	{attribute 'TcIecLibraryType'}
	{attribute 'external_name' := 'F_VN_RegionOrientationExp_GUID_B2683D61_49B5_467D_FA98_13B80F80665C'}
	(* Calculate the orientation of a region based on a binary image that contains a non zero value for every pixel in that region. (expert function) *)
	FUNCTION F_VN_RegionOrientationExp : HRESULT
	VAR_INPUT
		ipSrcImage	:	ITcVnImage;	(* Source image (1 channel, binary) *)
	END_VAR
	VAR_IN_OUT
		stOrientation	:	TcVnRotatedRectangle;	(* Resulting rotated rectangle, containig center of mass, lenghts of axes, and rotation angle of the region in clockwise direction. *)
	END_VAR
	VAR_INPUT
		eMethod	:	ETcVnOrientationMethod;	(* Method for calculating the orientation. *)
		hrPrev	:	HRESULT;	(* HRESULT indicating the result of previous operations (If SUCCEEDED(hrPrev) equals false, no operation is executed.) *)
	END_VAR

END_FUNCTION

// Functions/Measurement/F_VN_AdjustSearchWindowOrientationToLinearEdge

	{attribute 'TcIecLibraryType'}
	{attribute 'external_name' := 'F_VN_AdjustSearchWindowOrientationToLinearEdge_GUID_4BF80E17_9DF4_4449_FA19_D076489CDE34'}
	(* Adjust the search window to be orthogonal to a linear edge. Might be helpful before calling edge localization and distance measurement functions that rely on the search window. *)
	FUNCTION F_VN_AdjustSearchWindowOrientationToLinearEdge : HRESULT
	VAR_INPUT
		ipSrcImage	:	ITcVnImage;	(* Source image *)
	END_VAR
	VAR_IN_OUT
		aStartPoint	:	TcVnPoint2_REAL;	(* Position from which to start the search process (in the direction of aEndPoint), which is not changed *)
		aEndPoint	:	TcVnPoint2_REAL;	(* Position where the search process ends, which is adjusted by this function *)
	END_VAR
	VAR_INPUT
		eEdgeDirection	:	ETcVnEdgeDirection;	(* Specification of the edge direction to search for *)
		fMinStrength	:	REAL;	(* Specification of the minimum strength (intensity difference) of the edge to search for *)
		nMaxThickness	:	UDINT;	(* Specification of the maximum thickness of the edge to search for, which means fMinStrength must be reached within nMaxThickness pixels *)
		nSearchLines	:	UDINT;	(* Width of the search window, i.e. the number of search lines (3, 5, 7, ...), centered around the line specified by aStartPoint and aEndPoint *)
		hrPrev	:	HRESULT;	(* HRESULT indicating the result of previous operations (If SUCCEEDED(hrPrev) equals false, no operation is executed.) *)
	END_VAR

END_FUNCTION

// Functions/Measurement/F_VN_ClosestPointsBF

	{attribute 'TcIecLibraryType'}
	{attribute 'external_name' := 'F_VN_ClosestPointsBF_GUID_F8745723_FA66_485A_C6BC_8B3A81941337'}
	(* Find the closest distance between two 2d point sets of the same type, using a brute force approach. *)
	FUNCTION F_VN_ClosestPointsBF : HRESULT
	VAR_INPUT
		ipPointSet1	:	ITcVnContainer;	(* Container with 1st set of 2d points *)
		ipPointSet2	:	ITcVnContainer;	(* Container with 2nd set of 2d points *)
	END_VAR
	VAR_IN_OUT
		fMinDist	:	LREAL;	(* Returns the minimum distance between 2 points of the different point sets *)
		aPoint1	:	TcVnPoint2_LREAL;	(* Returns the point out of ipPointSet1, for which fMinDist is achieved *)
		aPoint2	:	TcVnPoint2_LREAL;	(* Returns the point out of ipPointSet2, for which fMinDist is achieved *)
	END_VAR
	VAR_INPUT
		hrPrev	:	HRESULT;	(* HRESULT indicating the result of previous operations (If SUCCEEDED(hrPrev) equals false, no operation is executed.) *)
	END_VAR

END_FUNCTION

// Functions/Measurement/F_VN_LocateCircularArc

	{attribute 'TcIecLibraryType'}
	{attribute 'external_name' := 'F_VN_LocateCircularArc_GUID_5C99AC69_8B36_49C3_F767_A0447ABA5FEC'}
	(* Locate a circular arc, using an interpolation method. *)
	FUNCTION F_VN_LocateCircularArc : HRESULT
	VAR_INPUT
		ipSrcImage	:	ITcVnImage;	(* Source image (1 channel) *)
	END_VAR
	VAR_IN_OUT
		stCircularArc	:	TcVnCircularArc;	(* Returns the circular arc parameters *)
		aCenter	:	TcVnPoint2_REAL;	(* Input estimated circle center (only used as a starting point to search for the circle contour, not used for the circle center estimation) *)
	END_VAR
	VAR_INPUT
		fSearchRadius	:	REAL;	(* Input search radius (starting from aCenter, should be greater than the actual circle radius but aCenter + fSearchRadius should be within the image borders) *)
		fArcDirectionRad	:	LREAL;	(* Input search starting direction in radian. Valid range is [-pi, +pi], where right is 0 rad, top is -pi/2 rad and bottom +pi/2 rad. The circular arc should at least be valid in range fArcDirectionRad +- 0.4 rad. *)
		eEdgeDirection	:	ETcVnEdgeDirection;	(* Specification of the edge direction to search for *)
		fMinStrength	:	REAL;	(* Specification of the minimum strength (intensity difference) of the edge to search for *)
		hrPrev	:	HRESULT;	(* HRESULT indicating the result of previous operations (If SUCCEEDED(hrPrev) equals false, no operation is executed.) *)
	END_VAR

END_FUNCTION

// Functions/Measurement/F_VN_LocateCircularArcExp

	{attribute 'TcIecLibraryType'}
	{attribute 'external_name' := 'F_VN_LocateCircularArcExp_GUID_D2973620_C78E_45B3_C257_FC79FEFA4F95'}
	(* Locate a circular arc. (expert function) *)
	FUNCTION F_VN_LocateCircularArcExp : HRESULT
	VAR_INPUT
		ipSrcImage	:	ITcVnImage;	(* Source image (1 channel) *)
	END_VAR
	VAR_IN_OUT
		stCircularArc	:	TcVnCircularArc;	(* Returns the circular arc parameters *)
		aCenter	:	TcVnPoint2_REAL;	(* Input estimated circle center (only used as a starting point to search for the circle contour, not used for the circle center estimation) *)
	END_VAR
	VAR_INPUT
		fSearchRadius	:	REAL;	(* Input search radius (starting from aCenter, should be greater than the actual circle radius but aCenter + fSearchRadius should be within the image borders) *)
		fArcDirectionRad	:	LREAL;	(* Input search starting direction in radian. Valid range is [-pi, +pi], where right is 0 rad, top is -pi/2 rad and bottom +pi/2 rad. The circular arc should at least be valid in range fArcDirectionRad +- 4 * fAngleStepRad) *)
		eEdgeDirection	:	ETcVnEdgeDirection;	(* Specification of the edge direction to search for *)
		fMinStrength	:	REAL;	(* Specification of the minimum strength (intensity difference) of the edge to search for *)
		fAngleStepRad	:	LREAL;	(* Search step in rad (should be chosen so that about 20 - 60 steps are available for the whole arc. In most cases 0.1 rad (5.7 deg) is a good value) *)
		nMaxThickness	:	UDINT;	(* Specification of the maximum thickness of the edge to search for, which means fMinStrength must be reached within nMaxThickness pixels *)
		bInvertSearchDirection	:	BOOL;	(* If true, the search starts from outside the circular arc in direction of the center *)
		nSubpixelsIterations	:	UDINT;	(* Specifies the number of subpixels (for INTERPOLATION, 10 - 20 usually is sufficient) or maximum number of iterations for optimizing the parameters (for APPROX_ERF and APPROX_GAUSSIAN, 50 - 100 usually is sufficient) *)
		fApproxPrecision	:	REAL;	(* Specifies the approximation precision for APPROX_ERF and APPROX_GAUSSIAN (0.001 usually is sufficient, unused for INTERPOLATION) *)
		eAlgorithm	:	ETcVnEdgeDetectionAlgorithm;	(* Selection of the edge detection algorithm *)
		ipContourPoints	:	REFERENCE TO ITcVnContainer;	(* Returns the subpixel accurate contour (optional, set to 0 if not required; ContainerType_Vector_TcVnPoint2_REAL; Non-zero interface pointers are reused.) *)
		hrPrev	:	HRESULT;	(* HRESULT indicating the result of previous operations (If SUCCEEDED(hrPrev) equals false, no operation is executed.) *)
	END_VAR

END_FUNCTION

// Functions/Measurement/F_VN_LocateEdge

	{attribute 'TcIecLibraryType'}
	{attribute 'external_name' := 'F_VN_LocateEdge_GUID_6D658DBC_9003_460D_D8DC_4EA5DD496210'}
	(* Locate the points of the first occuring edge inside a specified search window, using an interpolation method. *)
	FUNCTION F_VN_LocateEdge : HRESULT
	VAR_INPUT
		ipSrcImage	:	ITcVnImage;	(* Source image (1 channel) *)
		ipEdgePoints	:	REFERENCE TO ITcVnContainer;	(* Returns the detected edge points (ContainerType_Vector_TcVnPoint2_REAL) *)
	END_VAR
	VAR_IN_OUT
		aStartPoint	:	TcVnPoint2_REAL;	(* Position from which to start the search process (in the direction of aEndPoint) *)
		aEndPoint	:	TcVnPoint2_REAL;	(* Position where the search process ends *)
	END_VAR
	VAR_INPUT
		eEdgeDirection	:	ETcVnEdgeDirection;	(* Specification of the edge direction to search for *)
		fMinStrength	:	REAL;	(* Specification of the minimum strength (intensity difference) of the edge to search for *)
		nSearchLines	:	UDINT;	(* Width of the search window, i.e. the number of search lines (1, 3, 5, 7, ...), centered around the line specified by aStartPoint and aEndPoint *)
		hrPrev	:	HRESULT;	(* HRESULT indicating the result of previous operations (If SUCCEEDED(hrPrev) equals false, no operation is executed.) *)
	END_VAR
	VAR_OUTPUT
		fAvgStrength	:	REAL;	(* Returns the average strength of the detected edge *)
	END_VAR

END_FUNCTION

// Functions/Measurement/F_VN_LocateEdgeExp

	{attribute 'TcIecLibraryType'}
	{attribute 'external_name' := 'F_VN_LocateEdgeExp_GUID_71867877_E50C_46F9_ECC5_1606F0E48315'}
	(* Locate the points of the first occuring edge inside a specified search window with subpixel accuracy. (expert function) *)
	FUNCTION F_VN_LocateEdgeExp : HRESULT
	VAR_INPUT
		ipSrcImage	:	ITcVnImage;	(* Source image (1 channel) *)
		ipEdgePoints	:	REFERENCE TO ITcVnContainer;	(* Returns the detected edge points (ContainerType_Vector_TcVnPoint2_REAL) *)
	END_VAR
	VAR_IN_OUT
		aStartPoint	:	TcVnPoint2_REAL;	(* Position from which to start the search process (in the direction of aEndPoint) *)
		aEndPoint	:	TcVnPoint2_REAL;	(* Position where the search process ends *)
	END_VAR
	VAR_INPUT
		eEdgeDirection	:	ETcVnEdgeDirection;	(* Specification of the edge direction to search for *)
		fMinStrength	:	REAL;	(* Specification of the minimum strength (intensity difference) of the edge to search for *)
		nSearchLines	:	UDINT;	(* Width of the search window, i.e. the number of search lines (1, 3, 5, 7, ...), centered around the line specified by aStartPoint and aEndPoint *)
		fSearchLineDist	:	REAL;	(* Distance between the search lines in pixels (> 0) *)
		nMaxThickness	:	UDINT;	(* Specification of the maximum thickness of the edge to search for, which means fMinStrength must be reached within nMaxThickness pixels *)
		nSubpixelsIterations	:	UDINT;	(* Specifies the number of subpixels (for INTERPOLATION, 10 - 20 usually is sufficient) or maximum number of iterations for optimizing the parameters (for APPROX_ERF and APPROX_GAUSSIAN, 50 - 100 usually is sufficient) *)
		fApproxPrecision	:	REAL;	(* Specifies the approximation precision for APPROX_ERF and APPROX_GAUSSIAN (0.001 usually is sufficient, unused for INTERPOLATION) *)
		eAlgorithm	:	ETcVnEdgeDetectionAlgorithm;	(* Selection of the edge detection algorithm *)
		hrPrev	:	HRESULT;	(* HRESULT indicating the result of previous operations (If SUCCEEDED(hrPrev) equals false, no operation is executed.) *)
	END_VAR
	VAR_OUTPUT
		fAvgStrength	:	REAL;	(* Returns the average strength of the detected edge *)
	END_VAR

END_FUNCTION

// Functions/Measurement/F_VN_LocateEdges

	{attribute 'TcIecLibraryType'}
	{attribute 'external_name' := 'F_VN_LocateEdges_GUID_16CD5812_FF7D_41F8_D2D0_ABD474139878'}
	(* Locate the points of multiple occuring edges inside a specified search window, using an interpolation method. *)
	FUNCTION F_VN_LocateEdges : HRESULT
	VAR_INPUT
		ipSrcImage	:	ITcVnImage;	(* Source image (1 channel) *)
		ipEdgePoints	:	REFERENCE TO ITcVnContainer;	(* Returns the detected edge points (ContainerType_Vector_Vector_TcVnPoint2_REAL) *)
	END_VAR
	VAR_IN_OUT
		aStartPoint	:	TcVnPoint2_REAL;	(* Position from which to start the search process (in the direction of aEndPoint) *)
		aEndPoint	:	TcVnPoint2_REAL;	(* Position where the search process ends *)
	END_VAR
	VAR_INPUT
		nNumEdges	:	UDINT;	(* The (maximum) number of edges to search for *)
		eEdgeDirection	:	ETcVnEdgeDirection;	(* Specification of the edge direction to search for *)
		bAlternateDirection	:	BOOL;	(* If true, eEdgeDirection is alternated after each detected edge. Else, only edges with eEdgeDirection are searched for. *)
		fMinStrength	:	REAL;	(* Specification of the minimum strength (intensity difference) of the edge to search for *)
		nSearchLines	:	UDINT;	(* Width of the search window, i.e. the number of search lines (1, 3, 5, 7, ...), centered around the line specified by aStartPoint and aEndPoint *)
		hrPrev	:	HRESULT;	(* HRESULT indicating the result of previous operations (If SUCCEEDED(hrPrev) equals false, no operation is executed.) *)
	END_VAR
	VAR_OUTPUT
		fAvgStrength	:	REAL;	(* Returns the average strength of the detected edges *)
	END_VAR

END_FUNCTION

// Functions/Measurement/F_VN_LocateEdgesExp

	{attribute 'TcIecLibraryType'}
	{attribute 'external_name' := 'F_VN_LocateEdgesExp_GUID_24AB17DE_4502_4635_E826_7D952681F995'}
	(* Locate the points of multiple occuring edges inside a specified search window with subpixel accuracy. (expert function) *)
	FUNCTION F_VN_LocateEdgesExp : HRESULT
	VAR_INPUT
		ipSrcImage	:	ITcVnImage;	(* Source image (1 channel) *)
		ipEdgePoints	:	REFERENCE TO ITcVnContainer;	(* Returns the detected edge points (ContainerType_Vector_Vector_TcVnPoint2_REAL) *)
	END_VAR
	VAR_IN_OUT
		aStartPoint	:	TcVnPoint2_REAL;	(* Position from which to start the search process (in the direction of aEndPoint) *)
		aEndPoint	:	TcVnPoint2_REAL;	(* Position where the search process ends *)
	END_VAR
	VAR_INPUT
		nNumEdges	:	UDINT;	(* The (maximum) number of edges to search for *)
		eEdgeDirection	:	ETcVnEdgeDirection;	(* Specification of the edge direction to search for *)
		bAlternateDirection	:	BOOL;	(* If true, eEdgeDirection is alternated after each detected edge. Else, only edges with eEdgeDirection are searched for. *)
		fMinStrength	:	REAL;	(* Specification of the minimum strength (intensity difference) of the edge to search for *)
		nSearchLines	:	UDINT;	(* Width of the search window, i.e. the number of search lines (1, 3, 5, 7, ...), centered around the line specified by aStartPoint and aEndPoint *)
		fSearchLineDist	:	REAL;	(* Distance between the search lines in pixels (> 0) *)
		nMaxThickness	:	UDINT;	(* Specification of the maximum thickness of the edge to search for, which means fMinStrength must be reached within nMaxThickness pixels *)
		nSubpixelsIterations	:	UDINT;	(* Specifies the number of subpixels (for INTERPOLATION, 10 - 20 usually is sufficient) or maximum number of iterations for optimizing the parameters (for APPROX_ERF and APPROX_GAUSSIAN, 50 - 100 usually is sufficient) *)
		fApproxPrecision	:	REAL;	(* Specifies the approximation precision for APPROX_ERF and APPROX_GAUSSIAN (0.001 usually is sufficient, unused for INTERPOLATION) *)
		eAlgorithm	:	ETcVnEdgeDetectionAlgorithm;	(* Selection of the edge detection algorithm *)
		hrPrev	:	HRESULT;	(* HRESULT indicating the result of previous operations (If SUCCEEDED(hrPrev) equals false, no operation is executed.) *)
	END_VAR
	VAR_OUTPUT
		fAvgStrength	:	REAL;	(* Returns the average strength of the detected edges *)
	END_VAR

END_FUNCTION

// Functions/Measurement/F_VN_LocateEllipse

	{attribute 'TcIecLibraryType'}
	{attribute 'external_name' := 'F_VN_LocateEllipse_GUID_7D53F90F_C5F2_4037_E1F8_744121219137'}
	(* Locate an ellipse, using an interpolation method for locating the edges. *)
	FUNCTION F_VN_LocateEllipse : HRESULT
	VAR_INPUT
		ipSrcImage	:	ITcVnImage;	(* Source image (1 channel) *)
	END_VAR
	VAR_IN_OUT
		stEllipse	:	TcVnRotatedRectangle;	(* Returns the detected ellipse *)
		aCenter	:	TcVnPoint2_REAL;	(* The expected ellipse center *)
	END_VAR
	VAR_INPUT
		fSearchRadius	:	REAL;	(* Radius around aCenter to search for edges (aCenter + fSearchRadius in all directions must be inside image borders!) *)
		eEdgeDirection	:	ETcVnEdgeDirection;	(* Specification of the edge direction to search for (from center to outside ellipse) *)
		fMinStrength	:	REAL;	(* Specification of the minimum strength (intensity difference) of the edge to search for *)
		hrPrev	:	HRESULT;	(* HRESULT indicating the result of previous operations (If SUCCEEDED(hrPrev) equals false, no operation is executed.) *)
	END_VAR

END_FUNCTION

// Functions/Measurement/F_VN_LocateEllipseExp

	{attribute 'TcIecLibraryType'}
	{attribute 'external_name' := 'F_VN_LocateEllipseExp_GUID_0A60BF8D_B9F3_4F5C_FC58_D9258E827D64'}
	(* Locate an ellipse. (expert function) *)
	FUNCTION F_VN_LocateEllipseExp : HRESULT
	VAR_INPUT
		ipSrcImage	:	ITcVnImage;	(* Source image (1 channel) *)
	END_VAR
	VAR_IN_OUT
		stEllipse	:	TcVnRotatedRectangle;	(* Returns the detected ellipse *)
		aCenter	:	TcVnPoint2_REAL;	(* The expected ellipse center *)
	END_VAR
	VAR_INPUT
		fSearchRadius	:	REAL;	(* Radius around aCenter to search for edges *)
		eEdgeDirection	:	ETcVnEdgeDirection;	(* Specification of the edge direction to search for (from center to outside ellipse or other way round, if bInvertSearchDirection is true) *)
		fMinStrength	:	REAL;	(* Specification of the minimum strength (intensity difference) of the edge to search for *)
		nMaxThickness	:	UDINT;	(* Specification of the maximum thickness of the edge to search for, which means fMinStrength must be reached within nMaxThickness pixels *)
		bInvertSearchDirection	:	BOOL;	(* If true, the search starts from outside the ellipse in direction of the center *)
		fMinSearchRadius	:	REAL;	(* Radius around aCenter to skip before starting to search for edges (e.g. to save time or if the center contains edges that should be ignored) *)
		nSubpixelsIterations	:	UDINT;	(* Specifies the number of subpixels (for INTERPOLATION, 10 - 20 usually is sufficient) or maximum number of iterations for optimizing the parameters (for APPROX_ERF and APPROX_GAUSSIAN, 50 - 100 usually is sufficient) *)
		nSearchLines	:	UDINT;	(* Specifies the amount of search lines, which are equally distributed in all directions (must be >= 8 and a multiple of 4) *)
		fApproxPrecision	:	REAL;	(* Specifies the approximation precision for APPROX_ERF and APPROX_GAUSSIAN (0.001 usually is sufficient, unused for INTERPOLATION) *)
		eAlgorithm	:	ETcVnEdgeDetectionAlgorithm;	(* Selection of the edge detection algorithm *)
		ipContourPoints	:	REFERENCE TO ITcVnContainer;	(* Returns the subpixel accurate ellipse contour (optional, set to 0 if not required; ContainerType_Vector_TcVnPoint2_REAL; Non-zero interface pointers are reused.) *)
		hrPrev	:	HRESULT;	(* HRESULT indicating the result of previous operations (If SUCCEEDED(hrPrev) equals false, no operation is executed.) *)
	END_VAR

END_FUNCTION

// Functions/Measurement/F_VN_MeasureAngleBetweenEdges

	{attribute 'TcIecLibraryType'}
	{attribute 'external_name' := 'F_VN_MeasureAngleBetweenEdges_GUID_D045AAF4_339B_4CE5_F178_0EB747DFE41C'}
	(* Measure the angle between 2 edges, using an interpolation method. *)
	FUNCTION F_VN_MeasureAngleBetweenEdges : HRESULT
	VAR_INPUT
		ipSrcImage	:	ITcVnImage;	(* Source image (1 channel) *)
	END_VAR
	VAR_IN_OUT
		fAngle	:	REAL;	(* Returns the angle between the detected edges (radians) *)
		aInnerPoint	:	TcVnPoint2_REAL;	(* Position inside the angle to measure, from which to start the edge search process (in the direction of aOuterPoint1 and aOuterPoint2) *)
		aOuterPoint1	:	TcVnPoint2_REAL;	(* Position where the search process for edge 1 ends *)
		aOuterPoint2	:	TcVnPoint2_REAL;	(* Position where the search process for edge 2 ends *)
	END_VAR
	VAR_INPUT
		eEdgeDirection	:	ETcVnEdgeDirection;	(* Specification of the edge direction from aInnerPoint to aOuterPoint1 and aOuterPoint2 to search for *)
		fMinStrength	:	REAL;	(* Specification of the minimum strength (intensity difference) of the edge to search for *)
		nSearchLines	:	UDINT;	(* Width of the search windows, i.e. the number of search lines (3, 5, 7, ...), centered around the lines specified by aInnerPoint and aOuterPoint1, aOuterPoint2 *)
		hrPrev	:	HRESULT;	(* HRESULT indicating the result of previous operations (If SUCCEEDED(hrPrev) equals false, no operation is executed.) *)
	END_VAR

END_FUNCTION

// Functions/Measurement/F_VN_MeasureAngleBetweenEdgesExp

	{attribute 'TcIecLibraryType'}
	{attribute 'external_name' := 'F_VN_MeasureAngleBetweenEdgesExp_GUID_B9FC8105_DD76_4FBA_C762_CA24E7D135AD'}
	(* Measure the angle between 2 edges. *)
	FUNCTION F_VN_MeasureAngleBetweenEdgesExp : HRESULT
	VAR_INPUT
		ipSrcImage	:	ITcVnImage;	(* Source image (1 channel) *)
	END_VAR
	VAR_IN_OUT
		fAngle	:	REAL;	(* Returns the angle between the detected edges (radians or degrees, depending on bAngleInDegrees) *)
		aInnerPoint	:	TcVnPoint2_REAL;	(* Position inside the angle to measure, from which to start the edge search process (in the direction of aOuterPoint1 and aOuterPoint2) *)
		aOuterPoint1	:	TcVnPoint2_REAL;	(* Position where the search process for edge 1 ends *)
		aOuterPoint2	:	TcVnPoint2_REAL;	(* Position where the search process for edge 2 ends *)
	END_VAR
	VAR_INPUT
		eEdgeDirection	:	ETcVnEdgeDirection;	(* Specification of the edge direction from aInnerPoint to aOuterPoint1 and aOuterPoint2 to search for *)
		fMinStrength	:	REAL;	(* Specification of the minimum strength (intensity difference) of the edge to search for *)
		nSearchLines	:	UDINT;	(* Width of the search window, i.e. the number of search lines (3, 5, 7, ...), centered around the line specified by aInnerPoint and aOuterPoint1, aOuterPoint2 *)
		fSearchLineDist	:	REAL;	(* Distance between the search lines in pixels (> 0) *)
		nMaxThickness	:	UDINT;	(* Specification of the maximum thickness of the edge to search for, which means fMinStrength must be reached within nMaxThickness pixels *)
		bInvertSearchDirection	:	BOOL;	(* If true, the search starts from each aOuterPoint in direction of aInnerPoint *)
		nSubpixelsIterations	:	UDINT;	(* Specifies the number of subpixels (for INTERPOLATION, 10 - 20 usually is sufficient) or maximum number of iterations for optimizing the parameters (for APPROX_ERF and APPROX_GAUSSIAN, 50 - 100 usually is sufficient) *)
		bAngleInDegrees	:	BOOL;	(* fAngle is in degrees, if true *)
		fApproxPrecision	:	REAL;	(* Specifies the approximation precision for APPROX_ERF and APPROX_GAUSSIAN (0.001 usually is sufficient, unused for INTERPOLATION) *)
		eAlgorithm	:	ETcVnEdgeDetectionAlgorithm;	(* Selection of the edge detection algorithm *)
		ipEdgePoints1	:	REFERENCE TO ITcVnContainer;	(* Returns the detected edge points between aInnerPoint and aOuterPoint1 (ContainerType_Vector_TcVnPoint2_REAL) *)
		ipEdgePoints2	:	REFERENCE TO ITcVnContainer;	(* Returns the detected edge points between aInnerPoint and aOuterPoint2 (ContainerType_Vector_TcVnPoint2_REAL) *)
		hrPrev	:	HRESULT;	(* HRESULT indicating the result of previous operations (If SUCCEEDED(hrPrev) equals false, no operation is executed.) *)
	END_VAR

END_FUNCTION

// Functions/Measurement/F_VN_MeasureEdgeDistance

	{attribute 'TcIecLibraryType'}
	{attribute 'external_name' := 'F_VN_MeasureEdgeDistance_GUID_6B314BDA_9727_45F2_FABA_828BF07E8929'}
	(* Measure the distance between 2 parallel edges, using an interpolation method. *)
	FUNCTION F_VN_MeasureEdgeDistance : HRESULT
	VAR_INPUT
		ipSrcImage	:	ITcVnImage;	(* Source image (1 channel) *)
	END_VAR
	VAR_IN_OUT
		fAvgDistance	:	REAL;	(* Returns the average distance between the detected edges *)
		aStartPoint	:	TcVnPoint2_REAL;	(* Position from which to start the search process (in the direction of aEndPoint) *)
		aEndPoint	:	TcVnPoint2_REAL;	(* Position where the search process ends *)
	END_VAR
	VAR_INPUT
		eEdgeDirection	:	ETcVnEdgeDirection;	(* Specification of the edge direction from aStartPoint to aEndPoint to search for *)
		fMinStrength	:	REAL;	(* Specification of the minimum strength (intensity difference) of the edge to search for *)
		nSearchLines	:	UDINT;	(* Width of the search window, i.e. the number of search lines (1, 3, 5, 7, ...), centered around the line specified by aStartPoint and aEndPoint *)
		hrPrev	:	HRESULT;	(* HRESULT indicating the result of previous operations (If SUCCEEDED(hrPrev) equals false, no operation is executed.) *)
	END_VAR

END_FUNCTION

// Functions/Measurement/F_VN_MeasureEdgeDistanceExp

	{attribute 'TcIecLibraryType'}
	{attribute 'external_name' := 'F_VN_MeasureEdgeDistanceExp_GUID_B5A698E0_19B0_4B58_F68B_C2D607FA5C90'}
	(* Measure the distance between 2 parallel edges. (expert function) *)
	FUNCTION F_VN_MeasureEdgeDistanceExp : HRESULT
	VAR_INPUT
		ipSrcImage	:	ITcVnImage;	(* Source image (1 channel) *)
	END_VAR
	VAR_IN_OUT
		fAvgDistance	:	REAL;	(* Returns the average distance between the detected edges *)
		aStartPoint	:	TcVnPoint2_REAL;	(* Position from which to start the search process (in the direction of aEndPoint) *)
		aEndPoint	:	TcVnPoint2_REAL;	(* Position where the search process ends *)
	END_VAR
	VAR_INPUT
		eEdgeDirection	:	ETcVnEdgeDirection;	(* Specification of the edge direction from aStartPoint to aEndPoint to search for *)
		fMinStrength	:	REAL;	(* Specification of the minimum strength (intensity difference) of the edge to search for *)
		nSearchLines	:	UDINT;	(* Width of the search window, i.e. the number of search lines (1, 3, 5, 7, ...), centered around the line specified by aStartPoint and aEndPoint *)
		fSearchLineDist	:	REAL;	(* Distance between the search lines in pixels (> 0) *)
		nMaxThickness	:	UDINT;	(* Specification of the maximum thickness of the edge to search for, which means fMinStrength must be reached within nMaxThickness pixels *)
		bInvertSearchDirection	:	BOOL;	(* If true, the search starts from the center point between aStartPoint and aEndPoint in both directions *)
		fSearchGap	:	REAL;	(* Optional width of a gap (>= 0, centered between aStartPoint and aEndPoint), that is neglected for searching edges (can reduce execution time). The 2 edges to search for must be on different sides of the gap. *)
		nSubpixelsIterations	:	UDINT;	(* Specifies the number of subpixels (for INTERPOLATION, 10 - 20 usually is sufficient) or maximum number of iterations for optimizing the parameters (for APPROX_ERF and APPROX_GAUSSIAN, 50 - 100 usually is sufficient) *)
		fApproxPrecision	:	REAL;	(* Specifies the approximation precision for APPROX_ERF and APPROX_GAUSSIAN (0.001 usually is sufficient, unused for INTERPOLATION) *)
		eAlgorithm	:	ETcVnEdgeDetectionAlgorithm;	(* Selection of the edge detection algorithm *)
		ipEdgePoints1	:	REFERENCE TO ITcVnContainer;	(* Returns the detected edge points of the edge near aStartPoint (optional, set to 0 if not required; ContainerType_Vector_TcVnPoint2_REAL) *)
		ipEdgePoints2	:	REFERENCE TO ITcVnContainer;	(* Returns the detected edge points of the edge near aEndPoint (optional, set to 0 if not required; ContainerType_Vector_TcVnPoint2_REAL) *)
		ipDistances	:	REFERENCE TO ITcVnContainer;	(* Returns the distances between the detected edge points (optional, set to 0 if not required; ContainerType_Vector_REAL) *)
		hrPrev	:	HRESULT;	(* HRESULT indicating the result of previous operations (If SUCCEEDED(hrPrev) equals false, no operation is executed.) *)
	END_VAR

END_FUNCTION

// Functions/Measurement/F_VN_MeasureMinEdgeDistance

	{attribute 'TcIecLibraryType'}
	{attribute 'external_name' := 'F_VN_MeasureMinEdgeDistance_GUID_AD6515FF_4497_4F80_F2EC_1F853CD0ABA8'}
	(* Measure the minimum distance within the specified search window between 2 edges, using an interpolation method. *)
	FUNCTION F_VN_MeasureMinEdgeDistance : HRESULT
	VAR_INPUT
		ipSrcImage	:	ITcVnImage;	(* Source image (1 channel) *)
	END_VAR
	VAR_IN_OUT
		fMinDistance	:	REAL;	(* Returns the minimum distance between the detected edges *)
		aStartPoint	:	TcVnPoint2_REAL;	(* Position from which to start the search process (in the direction of aEndPoint) *)
		aEndPoint	:	TcVnPoint2_REAL;	(* Position where the search process ends *)
	END_VAR
	VAR_INPUT
		eEdgeDirection	:	ETcVnEdgeDirection;	(* Specification of the edge direction from aStartPoint to aEndPoint to search for *)
		fMinStrength	:	REAL;	(* Specification of the minimum strength (intensity difference) of the edge to search for *)
		nSearchLines	:	UDINT;	(* Width of the search window, i.e. the number of search lines (1, 3, 5, 7, ...), centered around the line specified by aStartPoint and aEndPoint *)
		hrPrev	:	HRESULT;	(* HRESULT indicating the result of previous operations (If SUCCEEDED(hrPrev) equals false, no operation is executed.) *)
	END_VAR

END_FUNCTION

// Functions/Measurement/F_VN_MeasureMinEdgeDistanceExp

	{attribute 'TcIecLibraryType'}
	{attribute 'external_name' := 'F_VN_MeasureMinEdgeDistanceExp_GUID_1BC885D6_665A_4846_FCF1_ACE60271C85F'}
	(* Measure the minimum distance within the specified search window between 2 edges. (expert function) *)
	FUNCTION F_VN_MeasureMinEdgeDistanceExp : HRESULT
	VAR_INPUT
		ipSrcImage	:	ITcVnImage;	(* Source image (1 channel) *)
	END_VAR
	VAR_IN_OUT
		fMinDistance	:	REAL;	(* Returns the minimum distance between the detected edges *)
		aStartPoint	:	TcVnPoint2_REAL;	(* Position from which to start the search process (in the direction of aEndPoint) *)
		aEndPoint	:	TcVnPoint2_REAL;	(* Position where the search process ends *)
	END_VAR
	VAR_INPUT
		eEdgeDirection	:	ETcVnEdgeDirection;	(* Specification of the edge direction from aStartPoint to aEndPoint to search for *)
		fMinStrength	:	REAL;	(* Specification of the minimum strength (intensity difference) of the edge to search for *)
		nSearchLines	:	UDINT;	(* Width of the search window, i.e. the number of search lines (1, 3, 5, 7, ...), centered around the line specified by aStartPoint and aEndPoint *)
		fSearchLineDist	:	REAL;	(* Distance between the search lines in pixels (> 0) *)
		nMaxThickness	:	UDINT;	(* Specification of the maximum thickness of the edge to search for, which means fMinStrength must be reached within nMaxThickness pixels *)
		bInvertSearchDirection	:	BOOL;	(* If true, the search starts from the center point between aStartPoint and aEndPoint in both directions *)
		fSearchGap	:	REAL;	(* Optional width of a gap (>= 0, centered between aStartPoint and aEndPoint), that is neglected for searching edges (can reduce execution time). The 2 edges to search for must be on different sides of the gap. *)
		nSubpixelsIterations	:	UDINT;	(* Specifies the number of subpixels (for INTERPOLATION, 10 - 20 usually is sufficient) or maximum number of iterations for optimizing the parameters (for APPROX_ERF and APPROX_GAUSSIAN, 50 - 100 usually is sufficient) *)
		fApproxPrecision	:	REAL;	(* Specifies the approximation precision for APPROX_ERF and APPROX_GAUSSIAN (0.001 usually is sufficient, unused for INTERPOLATION) *)
		eAlgorithm	:	ETcVnEdgeDetectionAlgorithm;	(* Selection of the edge detection algorithm *)
		ipEdgePoints1	:	REFERENCE TO ITcVnContainer;	(* Returns the detected edge points of the edge near aStartPoint (optional, set to 0 if not required; ContainerType_Vector_TcVnPoint2_REAL) *)
		ipEdgePoints2	:	REFERENCE TO ITcVnContainer;	(* Returns the detected edge points of the edge near aEndPoint (optional, set to 0 if not required; ContainerType_Vector_TcVnPoint2_REAL) *)
	END_VAR
	VAR_IN_OUT
		aPoint1	:	TcVnPoint2_REAL;	(* Returns the point on the edge near aStartPoint, for which the minimum distance is achieved *)
		aPoint2	:	TcVnPoint2_REAL;	(* Returns the point on the edge near aEndPoint, for which the minimum distance is achieved *)
	END_VAR
	VAR_INPUT
		hrPrev	:	HRESULT;	(* HRESULT indicating the result of previous operations (If SUCCEEDED(hrPrev) equals false, no operation is executed.) *)
	END_VAR

END_FUNCTION

// Functions/Basic Container Operations/F_VN_AdvanceIterator

	{attribute 'TcIecLibraryType'}
	{attribute 'external_name' := 'F_VN_AdvanceIterator_GUID_BB474257_49A1_491A_C59B_3A73BFBDADCD'}
	(* Advance an iterator by the specified offset. *)
	FUNCTION F_VN_AdvanceIterator : HRESULT
	VAR_INPUT
		ipIterator	:	ITcVnForwardIterator;	(* Iterator to be advanced *)
		nOffset	:	LINT;	(* Offset, by which ipIterator is advanced *)
		hrPrev	:	HRESULT;	(* HRESULT indicating the result of previous operations (If SUCCEEDED(hrPrev) equals false, no operation is executed.) *)
	END_VAR

END_FUNCTION

// Functions/Basic Container Operations/F_VN_CheckIfEmpty

	{attribute 'TcIecLibraryType'}
	{attribute 'external_name' := 'F_VN_CheckIfEmpty_GUID_E0A53B67_24F3_4293_F0BF_1138FF50B90F'}
	(* Checks if the container is empty. (Alternatively use interface method .CheckIfEmpty.) *)
	FUNCTION F_VN_CheckIfEmpty : HRESULT
	VAR_INPUT
		ipContainer	:	ITcVnContainer;	(* Container *)
		hrPrev	:	HRESULT;	(* HRESULT indicating the result of previous operations (If SUCCEEDED(hrPrev) equals false, no operation is executed.) *)
	END_VAR

END_FUNCTION

// Functions/Basic Container Operations/F_VN_CheckIfIteratorIsAtEnd

	{attribute 'TcIecLibraryType'}
	{attribute 'external_name' := 'F_VN_CheckIfIteratorIsAtEnd_GUID_274D6BDA_A18A_4220_EB37_904B12B4254C'}
	(* Checks if the iterator points to the past-the-end element. (Alternatively use interface method .CheckIfEnd.) *)
	FUNCTION F_VN_CheckIfIteratorIsAtEnd : HRESULT
	VAR_INPUT
		ipIterator	:	ITcVnForwardIterator;	(* Iterator *)
		hrPrev	:	HRESULT;	(* HRESULT indicating the result of previous operations (If SUCCEEDED(hrPrev) equals false, no operation is executed.) *)
	END_VAR

END_FUNCTION

// Functions/Basic Container Operations/F_VN_ConvertContainerType

	{attribute 'TcIecLibraryType'}
	{attribute 'external_name' := 'F_VN_ConvertContainerType_GUID_162E5640_4948_45CA_C1B0_AD4F8FA254D7'}
	(* Converts a container to another type (Struct element types are not supported). *)
	FUNCTION F_VN_ConvertContainerType : HRESULT
	VAR_INPUT
		ipSrcContainer	:	ITcVnContainer;	(* Source container *)
		ipDestContainer	:	REFERENCE TO ITcVnContainer;	(* Returns the converted container *)
		nDestTypeGuid	:	GUID;	(* Specifies the destination container type for the conversion *)
		hrPrev	:	HRESULT;	(* HRESULT indicating the result of previous operations (If SUCCEEDED(hrPrev) equals false, no operation is executed.) *)
	END_VAR

END_FUNCTION

// Functions/Basic Container Operations/F_VN_CopyContainer

	{attribute 'TcIecLibraryType'}
	{attribute 'external_name' := 'F_VN_CopyContainer_GUID_CD2C08EF_8FE6_4608_DF24_1DD6161E4D3C'}
	(* Copys a container. *)
	FUNCTION F_VN_CopyContainer : HRESULT
	VAR_INPUT
		ipSrcContainer	:	ITcVnContainer;	(* Source container *)
		ipDestContainer	:	REFERENCE TO ITcVnContainer;	(* Destination container (same type ID as ipSrcContainer; Non-zero interface pointers are reused.) *)
		hrPrev	:	HRESULT;	(* HRESULT indicating the result of previous operations (If SUCCEEDED(hrPrev) equals false, no operation is executed.) *)
	END_VAR

END_FUNCTION

// Functions/Basic Container Operations/F_VN_CopyContainerElementsConditional_ITcVnContainer

	{attribute 'TcIecLibraryType'}
	{attribute 'external_name' := 'F_VN_CopyContainerElementsConditional_ITcVnContainer_GUID_38C9E632_A344_46EF_EE90_9D4E506E1242'}
	(* Copys container elements to a new container, depending on a custom condition. *)
	FUNCTION F_VN_CopyContainerElementsConditional_ITcVnContainer : HRESULT
	VAR_INPUT
		ipSrcContainer	:	ITcVnContainer;	(* Source container *)
		ipDestContainer	:	REFERENCE TO ITcVnContainer;	(* Returns a container with elements, that match the condition *)
		ipConditionFB	:	ITcVnCustomElementCondition_ITcVnContainer;	(* Custom condition *)
		hrPrev	:	HRESULT;	(* HRESULT indicating the result of previous operations (If SUCCEEDED(hrPrev) equals false, no operation is executed.) *)
	END_VAR

END_FUNCTION

// Interfaces/Containers/Function Blocks/ITcVnCustomElementCondition_ITcVnContainer

	(* Offers an interface for a custom condition computed for a container. *)
	{attribute 'c++_compatible'}
	INTERFACE ITcVnCustomElementCondition_ITcVnContainer


(* Evaluates the condition for the container. *)
	{attribute 'c++_compatible'}
	{attribute 'minimal_input_size' := '4'}
	{attribute 'pack_mode' := '4'}
	METHOD Condition : BOOL
	VAR_INPUT
		ipElement : ITcVnContainer;
	END_VAR
END_METHOD

END_INTERFACE

// Functions/Basic Container Operations/F_VN_CopyContainerElementsConditional_ITcVnForwardIterator

	{attribute 'TcIecLibraryType'}
	{attribute 'external_name' := 'F_VN_CopyContainerElementsConditional_ITcVnForwardIterator_GUID_54D3BD23_7764_4082_E999_7E445C0C656A'}
	(* Copys container elements to a new container, depending on a custom condition. *)
	FUNCTION F_VN_CopyContainerElementsConditional_ITcVnForwardIterator : HRESULT
	VAR_INPUT
		ipSrcContainer	:	ITcVnContainer;	(* Source container *)
		ipDestContainer	:	REFERENCE TO ITcVnContainer;	(* Returns a container with elements, that match the condition *)
		ipConditionFB	:	ITcVnCustomElementCondition_ITcVnForwardIterator;	(* Custom condition *)
		hrPrev	:	HRESULT;	(* HRESULT indicating the result of previous operations (If SUCCEEDED(hrPrev) equals false, no operation is executed.) *)
	END_VAR

END_FUNCTION

// Interfaces/Containers/Function Blocks/ITcVnCustomElementCondition_ITcVnForwardIterator

	(* Offers an interface for a custom condition computed for an element represented by an ITcVnForwardIterator. *)
	{attribute 'c++_compatible'}
	INTERFACE ITcVnCustomElementCondition_ITcVnForwardIterator


(* Evaluates the condition for the provided element. *)
	{attribute 'c++_compatible'}
	{attribute 'minimal_input_size' := '4'}
	{attribute 'pack_mode' := '4'}
	METHOD Condition : BOOL
	VAR_INPUT
		ipElement : ITcVnForwardIterator;
	END_VAR
END_METHOD

END_INTERFACE

// Functions/Basic Container Operations/F_VN_CreateContainer

	{attribute 'TcIecLibraryType'}
	{attribute 'external_name' := 'F_VN_CreateContainer_GUID_765CD239_1B51_4265_F329_16D378364A1F'}
	(* Creates a container with type GUID nTypeGuid and return its container interface. *)
	FUNCTION F_VN_CreateContainer : HRESULT
	VAR_INPUT
		ipContainer	:	REFERENCE TO ITcVnContainer;	(* Returns the created container *)
		nTypeGuid	:	GUID;	(* Type GUID of the container to be created *)
		nElementNum	:	ULINT;	(* Number of elements *)
		hrPrev	:	HRESULT;	(* HRESULT indicating the result of previous operations (If SUCCEEDED(hrPrev) equals false, no operation is executed.) *)
	END_VAR

END_FUNCTION

// Functions/Basic Container Operations/F_VN_CreateContainerFromArray

	{attribute 'TcIecLibraryType'}
	{attribute 'external_name' := 'F_VN_CreateContainerFromArray_GUID_BDD496F5_D1ED_4E94_DAF9_EF87AC8540DE'}
	(* Creates a container with type GUID nTypeGuid, initialize it with provided data and return its container interface. Only supported for basic container types, i.e. not for containers of containers. *)
	FUNCTION F_VN_CreateContainerFromArray : HRESULT
	VAR_INPUT
		pData	:	PVOID;	(* Pointer to the data array. Make sure that the array contains at least nElementNum elements and that the array element type matches the container element type. *)
		ipContainer	:	REFERENCE TO ITcVnContainer;	(* Returns the created container *)
		nTypeGuid	:	GUID;	(* Type GUID of the container to be created *)
		nElementNum	:	ULINT;	(* Number of elements to copy from pData *)
		hrPrev	:	HRESULT;	(* HRESULT indicating the result of previous operations (If SUCCEEDED(hrPrev) equals false, no operation is executed.) *)
	END_VAR

END_FUNCTION

// Functions/Basic Container Operations/F_VN_EraseFromContainer

	{attribute 'TcIecLibraryType'}
	{attribute 'external_name' := 'F_VN_EraseFromContainer_GUID_C109E931_DF2B_4D22_F887_FD7297571336'}
	(* Erase elements from a container. *)
	FUNCTION F_VN_EraseFromContainer : HRESULT
	VAR_INPUT
		ipContainer	:	ITcVnContainer;	(* Container from which to erase elements *)
		nStartIdx	:	ULINT;	(* Index of the first element to erase *)
		nCount	:	ULINT;	(* Number of elements to erase *)
		hrPrev	:	HRESULT;	(* HRESULT indicating the result of previous operations (If SUCCEEDED(hrPrev) equals false, no operation is executed.) *)
	END_VAR

END_FUNCTION

// Functions/Basic Container Operations/F_VN_ExportContainer

	{attribute 'TcIecLibraryType'}
	{attribute 'external_name' := 'F_VN_ExportContainer_GUID_A49FF6C2_49C6_4CEB_CE9C_554167B375EE'}
	(* Export the container elements into a buffer (e.g. an array). Only possible for containers with basic elements. *)
	FUNCTION F_VN_ExportContainer : HRESULT
	VAR_INPUT
		ipContainer	:	ITcVnContainer;	(* Container with basic elements *)
		pBuffer	:	PVOID;	(* Buffer to store the container elements (Make sure to allocate enough memory! The required size in bytes can be determined using the function F_VN_ExportContainerSize) *)
		nBufferSize	:	ULINT;	(* Size of the buffer memory in bytes *)
		hrPrev	:	HRESULT;	(* HRESULT indicating the result of previous operations (If SUCCEEDED(hrPrev) equals false, no operation is executed.) *)
	END_VAR

END_FUNCTION

// Functions/Basic Container Operations/F_VN_ExportContainerSize

	{attribute 'TcIecLibraryType'}
	{attribute 'external_name' := 'F_VN_ExportContainerSize_GUID_617B109F_6B98_43A8_C39C_96EADF8478AE'}
	(* Determine the required buffer size in bytes to store all container elements (number_of_Elements * size_per_Element). Only possible for containers with basic elements. *)
	FUNCTION F_VN_ExportContainerSize : HRESULT
	VAR_INPUT
		ipContainer	:	ITcVnContainer;	(* Container with basic elements *)
	END_VAR
	VAR_IN_OUT
		nBufferSize	:	ULINT;	(* Output parameter containing the required buffer size *)
	END_VAR
	VAR_INPUT
		hrPrev	:	HRESULT;	(* HRESULT indicating the result of previous operations (If SUCCEEDED(hrPrev) equals false, no operation is executed.) *)
	END_VAR

END_FUNCTION

// Functions/Basic Container Operations/F_VN_ExportContainer_String

	{attribute 'TcIecLibraryType'}
	{attribute 'external_name' := 'F_VN_ExportContainer_String_GUID_4C5700EB_CAFD_4281_FADC_7EAE52F41D45'}
	(* Export the container elements into a string. Only possible for containers of type ContainerType_String_SINT. *)
	FUNCTION F_VN_ExportContainer_String : HRESULT
	VAR_INPUT
		ipContainer	:	ITcVnContainer;	(* Container of type ContainerType_String_SINT *)
	END_VAR
	VAR_IN_OUT CONSTANT
		sText	:	STRING;	(* Make sure to choose a sufficient STRING size! The required size can be determined using the function VnExportContainerSize. *)
	END_VAR
	VAR_INPUT
		nMaxLength	:	ULINT;	(* Maximum string length to export (including 0 termination). If the container content is longer, the string is cut off at nMaxLength - 1 and 0 termination is appended. In this case, S_FALSE is returned. *)
		hrPrev	:	HRESULT;	(* HRESULT indicating the result of previous operations (If SUCCEEDED(hrPrev) equals false, no operation is executed.) *)
	END_VAR

END_FUNCTION

// Functions/Basic Container Operations/F_VN_ExportSubContainer

	{attribute 'TcIecLibraryType'}
	{attribute 'external_name' := 'F_VN_ExportSubContainer_GUID_3BF97AA9_1C46_4E0E_EC11_2C43376095D7'}
	(* Export the container elements of a sub-container into a buffer (e.g. an array). Only possible for 2-dimensional containers with basic elements. *)
	FUNCTION F_VN_ExportSubContainer : HRESULT
	VAR_INPUT
		ipContainer	:	ITcVnContainer;	(* Container with basic elements *)
		nIndex	:	ULINT;	(* Index of the requested element *)
		pBuffer	:	PVOID;	(* Buffer to store the container elements (Make sure to allocate enough memory! The required size in bytes can be determined using the function F_VN_ExportSubContainerSize) *)
		nBufferSize	:	ULINT;	(* Size of the buffer memory in bytes *)
		hrPrev	:	HRESULT;	(* HRESULT indicating the result of previous operations (If SUCCEEDED(hrPrev) equals false, no operation is executed.) *)
	END_VAR

END_FUNCTION

// Functions/Basic Container Operations/F_VN_ExportSubContainerSize

	{attribute 'TcIecLibraryType'}
	{attribute 'external_name' := 'F_VN_ExportSubContainerSize_GUID_8DB82A59_EFD3_41AE_DD57_A33F94D54A67'}
	(* Determine the required buffer size in bytes to store all container elements of a sub-container (number_of_Elements * size_per_Element). Only possible for 2-dimensional containers with basic elements. *)
	FUNCTION F_VN_ExportSubContainerSize : HRESULT
	VAR_INPUT
		ipContainer	:	ITcVnContainer;	(* Container with basic elements *)
		nIndex	:	ULINT;	(* Index of the requested element *)
	END_VAR
	VAR_IN_OUT
		nBufferSize	:	ULINT;	(* Output parameter containing the required buffer size *)
	END_VAR
	VAR_INPUT
		hrPrev	:	HRESULT;	(* HRESULT indicating the result of previous operations (If SUCCEEDED(hrPrev) equals false, no operation is executed.) *)
	END_VAR

END_FUNCTION

// Functions/Basic Container Operations/F_VN_ExportSubContainer_String

	{attribute 'TcIecLibraryType'}
	{attribute 'external_name' := 'F_VN_ExportSubContainer_String_GUID_58DAF122_268B_4C9D_DE01_224D1BFA5CF8'}
	(* Export the container elements of a sub-container into a string. Only possible for 2-dimensional containers of type ContainerType_Vector_String_SINT. *)
	FUNCTION F_VN_ExportSubContainer_String : HRESULT
	VAR_INPUT
		ipContainer	:	ITcVnContainer;	(* Container of type ContainerType_Vector_String_SINT *)
		nIndex	:	ULINT;	(* Index of the requested element *)
	END_VAR
	VAR_IN_OUT CONSTANT
		sText	:	STRING;	(* Make sure to choose a sufficient STRING size! The required size can be determined using the function VnExportSubContainerSize. *)
	END_VAR
	VAR_INPUT
		nMaxLength	:	ULINT;	(* Maximum string length to export (including 0 termination). If the container content is longer, the string is cut off at nMaxLength - 1 and 0 termination is appended. In this case, S_FALSE is returned. *)
		hrPrev	:	HRESULT;	(* HRESULT indicating the result of previous operations (If SUCCEEDED(hrPrev) equals false, no operation is executed.) *)
	END_VAR

END_FUNCTION

// Functions/Basic Container Operations/F_VN_ExtractContainerRange

	{attribute 'TcIecLibraryType'}
	{attribute 'external_name' := 'F_VN_ExtractContainerRange_GUID_593D2FC2_DA0F_4836_FDE3_513BE15EBB7F'}
	(* Copy the specified range of the source container into the destination container. (If the destination container already contains elements, they will be removed.) *)
	FUNCTION F_VN_ExtractContainerRange : HRESULT
	VAR_INPUT
		ipSrcContainer	:	ITcVnContainer;	(* Source container *)
		ipDestContainer	:	REFERENCE TO ITcVnContainer;	(* Destination container *)
		nFirstIdx	:	ULINT;	(* Index of the first element to copy *)
		nLastIdx	:	ULINT;	(* Index of the last element to copy *)
		hrPrev	:	HRESULT;	(* HRESULT indicating the result of previous operations (If SUCCEEDED(hrPrev) equals false, no operation is executed.) *)
	END_VAR

END_FUNCTION

// Functions/Basic Container Operations/F_VN_GetContainer

	{attribute 'TcIecLibraryType'}
	{attribute 'external_name' := 'F_VN_GetContainer_GUID_30DFF044_4FF2_4DD8_FBE7_B41FD65C96D4'}
	(* Gets a pointer to the current element converted into an ITcVnContainer interface and increment its reference counter (only possible for container types). (Alternatively use interface method .GetContainer.) *)
	FUNCTION F_VN_GetContainer : HRESULT
	VAR_INPUT
		ipIterator	:	ITcVnForwardIterator;	(* Iterator *)
		ipContainer	:	REFERENCE TO ITcVnContainer;	(* Returns the container interface *)
		hrPrev	:	HRESULT;	(* HRESULT indicating the result of previous operations (If SUCCEEDED(hrPrev) equals false, no operation is executed.) *)
	END_VAR

END_FUNCTION

// Functions/Basic Container Operations/F_VN_GetContainerExp

	{attribute 'TcIecLibraryType'}
	{attribute 'external_name' := 'F_VN_GetContainerExp_GUID_54E35AC9_220F_4D66_D127_BFD27CFBE634'}
	(* Gets a pointer to the current element converted into an ITcVnContainer interface and increment its reference counter (only possible for container types). Additionally, an offset to increment or decrement the iterator afterwards can be provided. (expert function) *)
	FUNCTION F_VN_GetContainerExp : HRESULT
	VAR_INPUT
		ipIterator	:	ITcVnForwardIterator;	(* Iterator *)
		ipContainer	:	REFERENCE TO ITcVnContainer;	(* Returns the container interface *)
		nOffset	:	DINT;	(* Offset to increment (>0) or decrement (<0) the iterator afterwards *)
		hrPrev	:	HRESULT;	(* HRESULT indicating the result of previous operations (If SUCCEEDED(hrPrev) equals false, no operation is executed.) *)
	END_VAR

END_FUNCTION

// Functions/Basic Container Operations/F_VN_GetForwardIterator

	{attribute 'TcIecLibraryType'}
	{attribute 'external_name' := 'F_VN_GetForwardIterator_GUID_5488245A_86ED_4BC6_E87B_8C5C2209F57D'}
	(* Gets a forward iterator for the container. (Alternatively use interface method .GetForwardIterator.) *)
	FUNCTION F_VN_GetForwardIterator : HRESULT
	VAR_INPUT
		ipContainer	:	ITcVnContainer;	(* Container *)
		ipIterator	:	REFERENCE TO ITcVnForwardIterator;	(* Returns the iterator interface *)
		hrPrev	:	HRESULT;	(* HRESULT indicating the result of previous operations (If SUCCEEDED(hrPrev) equals false, no operation is executed.) *)
	END_VAR

END_FUNCTION

// Functions/Basic Container Operations/F_VN_GetNumberOfElements

	{attribute 'TcIecLibraryType'}
	{attribute 'external_name' := 'F_VN_GetNumberOfElements_GUID_D6E7E122_1A05_4C7A_DB7C_0ED7F6ECC836'}
	(* Gets the number of elements in the container. (Alternatively use interface method .getElementNum.) *)
	FUNCTION F_VN_GetNumberOfElements : HRESULT
	VAR_INPUT
		ipContainer	:	ITcVnContainer;	(* Container *)
	END_VAR
	VAR_IN_OUT
		nNumberOfElements	:	ULINT;	(* Returns the number of elements in ipContainer *)
	END_VAR
	VAR_INPUT
		hrPrev	:	HRESULT;	(* HRESULT indicating the result of previous operations (If SUCCEEDED(hrPrev) equals false, no operation is executed.) *)
	END_VAR

END_FUNCTION

// Functions/Basic Container Operations/F_VN_GetRandomAccessIterator

	{attribute 'TcIecLibraryType'}
	{attribute 'external_name' := 'F_VN_GetRandomAccessIterator_GUID_2826886A_B6B4_469F_DEFD_12E791BA3D78'}
	(* Gets a random access iterator for the container. (Alternatively use interface method .GetRandomAccessIterator.) *)
	FUNCTION F_VN_GetRandomAccessIterator : HRESULT
	VAR_INPUT
		ipContainer	:	ITcVnContainer;	(* Container *)
		ipIterator	:	REFERENCE TO ITcVnRandomAccessIterator;	(* Returns the iterator interface *)
		hrPrev	:	HRESULT;	(* HRESULT indicating the result of previous operations (If SUCCEEDED(hrPrev) equals false, no operation is executed.) *)
	END_VAR

END_FUNCTION

// Functions/Basic Container Operations/F_VN_IncrementIterator

	{attribute 'TcIecLibraryType'}
	{attribute 'external_name' := 'F_VN_IncrementIterator_GUID_7E2EC18C_8E09_403B_CEFA_AD1C19772E7B'}
	(* Increment the iterator. (Alternatively use interface method .Increment.) *)
	FUNCTION F_VN_IncrementIterator : HRESULT
	VAR_INPUT
		ipIterator	:	ITcVnForwardIterator;	(* Iterator *)
		hrPrev	:	HRESULT;	(* HRESULT indicating the result of previous operations (If SUCCEEDED(hrPrev) equals false, no operation is executed.) *)
	END_VAR

END_FUNCTION

// Functions/Basic Container Operations/F_VN_IteratorDistance

	{attribute 'TcIecLibraryType'}
	{attribute 'external_name' := 'F_VN_IteratorDistance_GUID_CB9F9201_A839_4260_F1F3_E9E16F33E7ED'}
	(* Computes the distance between 2 iterators. *)
	FUNCTION F_VN_IteratorDistance : HRESULT
	VAR_INPUT
		ipIteratorFirst	:	ITcVnForwardIterator;	(* First iterator *)
		ipIteratorLast	:	ITcVnForwardIterator;	(* Last iterator *)
	END_VAR
	VAR_IN_OUT
		nDistance	:	LINT;	(* Returns the computed distance *)
	END_VAR
	VAR_INPUT
		hrPrev	:	HRESULT;	(* HRESULT indicating the result of previous operations (If SUCCEEDED(hrPrev) equals false, no operation is executed.) *)
	END_VAR

END_FUNCTION

// Functions/Basic Container Operations/F_VN_ReserveContainerMemory

	{attribute 'TcIecLibraryType'}
	{attribute 'external_name' := 'F_VN_ReserveContainerMemory_GUID_B146C93C_8BCD_43A4_C31E_5B3577944643'}
	(* Reserve container memory (call with maximum required number of elements before manually appending elements for better performance) *)
	FUNCTION F_VN_ReserveContainerMemory : HRESULT
	VAR_INPUT
		ipContainer	:	ITcVnContainer;	(* Container for which to reserve the memory *)
		nElements	:	ULINT;	(* Number of elements for which the container should reserve memory *)
		hrPrev	:	HRESULT;	(* HRESULT indicating the result of previous operations (If SUCCEEDED(hrPrev) equals false, no operation is executed.) *)
	END_VAR

END_FUNCTION

// Functions/Basic Container Operations/F_VN_ReverseContainer

	{attribute 'TcIecLibraryType'}
	{attribute 'external_name' := 'F_VN_ReverseContainer_GUID_227EB9CF_E921_4E30_F557_D6286754B0CD'}
	(* Reverse the container elements. *)
	FUNCTION F_VN_ReverseContainer : HRESULT
	VAR_INPUT
		ipContainer	:	ITcVnContainer;	(* Container to be reversed *)
		hrPrev	:	HRESULT;	(* HRESULT indicating the result of previous operations (If SUCCEEDED(hrPrev) equals false, no operation is executed.) *)
	END_VAR

END_FUNCTION

// Functions/Basic Container Operations/F_VN_SetContainer

	{attribute 'TcIecLibraryType'}
	{attribute 'external_name' := 'F_VN_SetContainer_GUID_F41CD10F_04D0_4C1E_D76C_E282188D6FCD'}
	(* Sets the current element using an ITcVnContainer interface (only possible for container types). (Alternatively use interface method .SetContainer.) *)
	FUNCTION F_VN_SetContainer : HRESULT
	VAR_INPUT
		ipIterator	:	ITcVnForwardIterator;	(* Iterator *)
		ipContainer	:	ITcVnContainer;	(* Container interface of which the content is to be assigned to the current element *)
		hrPrev	:	HRESULT;	(* HRESULT indicating the result of previous operations (If SUCCEEDED(hrPrev) equals false, no operation is executed.) *)
	END_VAR

END_FUNCTION

// Functions/Basic Container Operations/F_VN_SetIteratorToBegin

	{attribute 'TcIecLibraryType'}
	{attribute 'external_name' := 'F_VN_SetIteratorToBegin_GUID_466B73A3_3F4B_4076_E4EE_02DCA3C37125'}
	(* Sets the iterator to the first element of the container. (Alternatively use interface method .SetToBegin.) *)
	FUNCTION F_VN_SetIteratorToBegin : HRESULT
	VAR_INPUT
		ipIterator	:	ITcVnForwardIterator;	(* Iterator *)
		hrPrev	:	HRESULT;	(* HRESULT indicating the result of previous operations (If SUCCEEDED(hrPrev) equals false, no operation is executed.) *)
	END_VAR

END_FUNCTION

// Functions/Geometric and Coordinate Transformations/F_VN_AlignRotatedImageRegion

	{attribute 'TcIecLibraryType'}
	{attribute 'external_name' := 'F_VN_AlignRotatedImageRegion_GUID_28A9F4C0_6F92_44FA_E782_CD76620100CF'}
	(* Copies the provided image region and aligns it to the image axes. *)
	FUNCTION F_VN_AlignRotatedImageRegion : HRESULT
	VAR_INPUT
		ipSrcImage	:	ITcVnImage;	(* Source image *)
		ipDestImage	:	REFERENCE TO ITcVnImage;	(* Destination image (An appropriate image will be created if required.) *)
	END_VAR
	VAR_IN_OUT
		stRegion	:	TcVnRotatedRectangle;	(* Image region to be aligned *)
	END_VAR
	VAR_INPUT
		hrPrev	:	HRESULT;	(* HRESULT indicating the result of previous operations (If SUCCEEDED(hrPrev) equals false, no operation is executed.) *)
	END_VAR

END_FUNCTION

// Functions/Geometric and Coordinate Transformations/F_VN_AlignRotatedImageRegionExp

	{attribute 'TcIecLibraryType'}
	{attribute 'external_name' := 'F_VN_AlignRotatedImageRegionExp_GUID_C4B5F369_F050_45D1_CE91_B306699607DF'}
	(* Copies the provided image region and aligns it to the image axes. (expert function) *)
	FUNCTION F_VN_AlignRotatedImageRegionExp : HRESULT
	VAR_INPUT
		ipSrcImage	:	ITcVnImage;	(* Source image *)
		ipDestImage	:	REFERENCE TO ITcVnImage;	(* Destination image (An appropriate image will be created if required.) *)
	END_VAR
	VAR_IN_OUT
		stRegion	:	TcVnRotatedRectangle;	(* Image region to be aligned *)
	END_VAR
	VAR_INPUT
		eInterpolationType	:	ETcVnInterpolationType;	(* Interpolation method *)
		eBorderInterpolation	:	ETcVnBorderInterpolationMethod;	(* Border interpolation method (ISOLATED not supported) *)
	END_VAR
	VAR_IN_OUT
		aBorderValue	:	TcVnVector4_LREAL;	(* Border value, if CONSTANT is used *)
	END_VAR
	VAR_INPUT
		hrPrev	:	HRESULT;	(* HRESULT indicating the result of previous operations (If SUCCEEDED(hrPrev) equals false, no operation is executed.) *)
	END_VAR

END_FUNCTION

// Functions/Geometric and Coordinate Transformations/F_VN_ApplyRotationToAffineTransformation

	{attribute 'TcIecLibraryType'}
	{attribute 'external_name' := 'F_VN_ApplyRotationToAffineTransformation_GUID_C5254176_148F_48F3_C7A7_2544A40C33EC'}
	(* Apply a rotation to an existing 2D affine transformation matrix. *)
	FUNCTION F_VN_ApplyRotationToAffineTransformation : HRESULT
	VAR_IN_OUT
		aTransformationMatrix	:	TcVnMatrix2x3_LREAL;	(* Affine transformation matrix to which the rotation is applied *)
	END_VAR
	VAR_INPUT
		fAngle	:	LREAL;	(* Angle in radians (positive means counter-clockwise) *)
		hrPrev	:	HRESULT;	(* HRESULT indicating the result of previous operations (If SUCCEEDED(hrPrev) equals false, no operation is executed.) *)
	END_VAR

END_FUNCTION

// Functions/Geometric and Coordinate Transformations/F_VN_ApplyRotationToAffineTransformationExp

	{attribute 'TcIecLibraryType'}
	{attribute 'external_name' := 'F_VN_ApplyRotationToAffineTransformationExp_GUID_1E0EBA39_528D_4A10_D427_D64732ACA9B4'}
	(* Apply a rotation to an existing 2D affine transformation matrix. (expert function) *)
	FUNCTION F_VN_ApplyRotationToAffineTransformationExp : HRESULT
	VAR_IN_OUT
		aTransformationMatrix	:	TcVnMatrix2x3_LREAL;	(* Affine transformation matrix to which the rotation is applied *)
	END_VAR
	VAR_INPUT
		fAngle	:	LREAL;	(* Angle in radians (positive means counter-clockwise) *)
		bUsePreMultiplication	:	BOOL;	(* Select if pre- or post-multiplication should be used *)
		hrPrev	:	HRESULT;	(* HRESULT indicating the result of previous operations (If SUCCEEDED(hrPrev) equals false, no operation is executed.) *)
	END_VAR

END_FUNCTION

// Functions/Geometric and Coordinate Transformations/F_VN_ApplyScalingToAffineTransformation

	{attribute 'TcIecLibraryType'}
	{attribute 'external_name' := 'F_VN_ApplyScalingToAffineTransformation_GUID_1D4CDC2B_D8C1_4D9C_D702_AEFDC573D0EB'}
	(* Apply a scaling to an existing 2D affine transformation matrix. *)
	FUNCTION F_VN_ApplyScalingToAffineTransformation : HRESULT
	VAR_IN_OUT
		aTransformationMatrix	:	TcVnMatrix2x3_LREAL;	(* Affine transformation matrix to which the scaling is applied *)
	END_VAR
	VAR_INPUT
		fScaleX	:	LREAL;	(* Scaling factor in x direction *)
		fScaleY	:	LREAL;	(* Scaling factor in y direction *)
		hrPrev	:	HRESULT;	(* HRESULT indicating the result of previous operations (If SUCCEEDED(hrPrev) equals false, no operation is executed.) *)
	END_VAR

END_FUNCTION

// Functions/Geometric and Coordinate Transformations/F_VN_ApplyScalingToAffineTransformationExp

	{attribute 'TcIecLibraryType'}
	{attribute 'external_name' := 'F_VN_ApplyScalingToAffineTransformationExp_GUID_1C9266A4_B171_46CC_EAD0_F36F20191B42'}
	(* Apply a scaling to an existing 2D affine transformation matrix. (expert function) *)
	FUNCTION F_VN_ApplyScalingToAffineTransformationExp : HRESULT
	VAR_IN_OUT
		aTransformationMatrix	:	TcVnMatrix2x3_LREAL;	(* Affine transformation matrix to which the scaling is applied *)
	END_VAR
	VAR_INPUT
		fScaleX	:	LREAL;	(* Scaling factor in x direction *)
		fScaleY	:	LREAL;	(* Scaling factor in y direction *)
		bUsePreMultiplication	:	BOOL;	(* Select if pre- or post-multiplication should be used *)
		hrPrev	:	HRESULT;	(* HRESULT indicating the result of previous operations (If SUCCEEDED(hrPrev) equals false, no operation is executed.) *)
	END_VAR

END_FUNCTION

// Functions/Geometric and Coordinate Transformations/F_VN_ApplyTranslationToAffineTransformation

	{attribute 'TcIecLibraryType'}
	{attribute 'external_name' := 'F_VN_ApplyTranslationToAffineTransformation_GUID_3B6C9DFC_5EAA_43EC_D3FD_036A0F2BAFC3'}
	(* Apply a translation to an existing 2D affine transformation matrix. *)
	FUNCTION F_VN_ApplyTranslationToAffineTransformation : HRESULT
	VAR_IN_OUT
		aTransformationMatrix	:	TcVnMatrix2x3_LREAL;	(* Affine transformation matrix to which the translation is applied *)
	END_VAR
	VAR_INPUT
		fDeltaX	:	LREAL;	(* Translation in x direction *)
		fDeltaY	:	LREAL;	(* Translation in y direction *)
		hrPrev	:	HRESULT;	(* HRESULT indicating the result of previous operations (If SUCCEEDED(hrPrev) equals false, no operation is executed.) *)
	END_VAR

END_FUNCTION

// Functions/Geometric and Coordinate Transformations/F_VN_ApplyTranslationToAffineTransformationExp

	{attribute 'TcIecLibraryType'}
	{attribute 'external_name' := 'F_VN_ApplyTranslationToAffineTransformationExp_GUID_A301A846_2E2C_48C0_DBAE_5B7B748A86F6'}
	(* Apply a translation to an existing 2D affine transformation matrix. (expert function) *)
	FUNCTION F_VN_ApplyTranslationToAffineTransformationExp : HRESULT
	VAR_IN_OUT
		aTransformationMatrix	:	TcVnMatrix2x3_LREAL;	(* Affine transformation matrix to which the translation is applied *)
	END_VAR
	VAR_INPUT
		fDeltaX	:	LREAL;	(* Translation in x direction *)
		fDeltaY	:	LREAL;	(* Translation in y direction *)
		bUsePreMultiplication	:	BOOL;	(* Select if pre- or post-multiplication should be used *)
		hrPrev	:	HRESULT;	(* HRESULT indicating the result of previous operations (If SUCCEEDED(hrPrev) equals false, no operation is executed.) *)
	END_VAR

END_FUNCTION

// Functions/Geometric and Coordinate Transformations/F_VN_ApplyYAxisInversionToAffineTransformation

	{attribute 'TcIecLibraryType'}
	{attribute 'external_name' := 'F_VN_ApplyYAxisInversionToAffineTransformation_GUID_BC281208_DFD9_4B72_E5D1_A38D0FD1606C'}
	(* Apply an inversion of the y-axis direction to an existing 2D affine transformation matrix. *)
	FUNCTION F_VN_ApplyYAxisInversionToAffineTransformation : HRESULT
	VAR_IN_OUT
		aTransformationMatrix	:	TcVnMatrix2x3_LREAL;	(* Affine transformation matrix to which the inversion of the y-axis direction is applied *)
	END_VAR
	VAR_INPUT
		hrPrev	:	HRESULT;	(* HRESULT indicating the result of previous operations (If SUCCEEDED(hrPrev) equals false, no operation is executed.) *)
	END_VAR

END_FUNCTION

// Functions/Geometric and Coordinate Transformations/F_VN_ApplyYAxisInversionToAffineTransformationExp

	{attribute 'TcIecLibraryType'}
	{attribute 'external_name' := 'F_VN_ApplyYAxisInversionToAffineTransformationExp_GUID_12969EA6_FE3A_4698_C3EB_534BE136C46B'}
	(* Apply an inversion of the y-axis direction to an existing 2D affine transformation matrix. (expert function) *)
	FUNCTION F_VN_ApplyYAxisInversionToAffineTransformationExp : HRESULT
	VAR_IN_OUT
		aTransformationMatrix	:	TcVnMatrix2x3_LREAL;	(* Affine transformation matrix to which the inversion of the y-axis direction is applied *)
	END_VAR
	VAR_INPUT
		bUsePreMultiplication	:	BOOL;	(* Select if pre- or post-multiplication should be used *)
		hrPrev	:	HRESULT;	(* HRESULT indicating the result of previous operations (If SUCCEEDED(hrPrev) equals false, no operation is executed.) *)
	END_VAR

END_FUNCTION

// Functions/Geometric and Coordinate Transformations/F_VN_ConvertCartesianToPolarAngleImage

	{attribute 'TcIecLibraryType'}
	{attribute 'external_name' := 'F_VN_ConvertCartesianToPolarAngleImage_GUID_00657097_243E_42BA_FC71_E412CBEBC36B'}
	(* Converts cartesian coordinates (x, y) to polar angle. *)
	FUNCTION F_VN_ConvertCartesianToPolarAngleImage : HRESULT
	VAR_INPUT
		ipSrcImageX	:	ITcVnImage;	(* Source image containing the x values (elements of type REAL or LREAL) *)
		ipSrcImageY	:	ITcVnImage;	(* Source image containing the y values (Same element type as ipSrcImageX) *)
		ipDestImageAng	:	REFERENCE TO ITcVnImage;	(* Destination image containing the angles (Same element type as source images. An appropriate destination image will be created if required.) *)
		hrPrev	:	HRESULT;	(* HRESULT indicating the result of previous operations (If SUCCEEDED(hrPrev) equals false, no operation is executed.) *)
	END_VAR

END_FUNCTION

// Functions/Geometric and Coordinate Transformations/F_VN_ConvertCartesianToPolarAngleImageExp

	{attribute 'TcIecLibraryType'}
	{attribute 'external_name' := 'F_VN_ConvertCartesianToPolarAngleImageExp_GUID_0AE7DF51_FBB3_476D_F829_C2661981E7F0'}
	(* Converts cartesian coordinates (x, y) to polar angle. (expert function) *)
	FUNCTION F_VN_ConvertCartesianToPolarAngleImageExp : HRESULT
	VAR_INPUT
		ipSrcImageX	:	ITcVnImage;	(* Source image containing the x values (elements of type REAL or LREAL) *)
		ipSrcImageY	:	ITcVnImage;	(* Source image containing the y values (Same element type as ipSrcImageX) *)
		ipDestImageAng	:	REFERENCE TO ITcVnImage;	(* Destination image containing the angles (Same element type as source images. An appropriate destination image will be created if required.) *)
		bAngleInDegrees	:	BOOL;	(* Specifys, if the angles should be in degrees or radians *)
		hrPrev	:	HRESULT;	(* HRESULT indicating the result of previous operations (If SUCCEEDED(hrPrev) equals false, no operation is executed.) *)
	END_VAR

END_FUNCTION

// Functions/Geometric and Coordinate Transformations/F_VN_ConvertCartesianToPolarAngles

	{attribute 'TcIecLibraryType'}
	{attribute 'external_name' := 'F_VN_ConvertCartesianToPolarAngles_GUID_F09BE09D_C276_43F7_C49B_0B521276F231'}
	(* Converts cartesian coordinates (x, y) to polar angle. *)
	FUNCTION F_VN_ConvertCartesianToPolarAngles : HRESULT
	VAR_INPUT
		ipSrcPointsCart	:	ITcVnContainer;	(* Container with cartesian points (ContainerType_Vector_TcVnPoint2_DINT or ContainerType_Vector_TcVnPoint2_REAL or ContainerType_Vector_TcVnPoint2_LREAL) *)
		ipDestAngles	:	REFERENCE TO ITcVnContainer;	(* Returns a container which is filled with the angles (ContainerType_Vector_REAL, if source points are of type TcVnPoint2_DINT or TcVnPoint2_REAL; else ContainerType_Vector_LREAL. Non-zero interface pointers are reused.) *)
		hrPrev	:	HRESULT;	(* HRESULT indicating the result of previous operations (If SUCCEEDED(hrPrev) equals false, no operation is executed.) *)
	END_VAR

END_FUNCTION

// Functions/Geometric and Coordinate Transformations/F_VN_ConvertCartesianToPolarAnglesExp

	{attribute 'TcIecLibraryType'}
	{attribute 'external_name' := 'F_VN_ConvertCartesianToPolarAnglesExp_GUID_469B1394_0CA6_44F4_C764_DB6342145354'}
	(* Converts cartesian coordinates (x, y) to polar angle. (expert function) *)
	FUNCTION F_VN_ConvertCartesianToPolarAnglesExp : HRESULT
	VAR_INPUT
		ipSrcPointsCart	:	ITcVnContainer;	(* Container with cartesian points (ContainerType_Vector_TcVnPoint2_DINT or ContainerType_Vector_TcVnPoint2_REAL or ContainerType_Vector_TcVnPoint2_LREAL) *)
		ipDestAngles	:	REFERENCE TO ITcVnContainer;	(* Returns a container which is filled with the angles (ContainerType_Vector_REAL, if source points are of type TcVnPoint2_DINT or TcVnPoint2_REAL; else ContainerType_Vector_LREAL. Non-zero interface pointers are reused.) *)
		bAngleInDegrees	:	BOOL;	(* Specify, if the angles should be in degrees or radians *)
		hrPrev	:	HRESULT;	(* HRESULT indicating the result of previous operations (If SUCCEEDED(hrPrev) equals false, no operation is executed.) *)
	END_VAR

END_FUNCTION

// Functions/Geometric and Coordinate Transformations/F_VN_ConvertCartesianToPolarImages

	{attribute 'TcIecLibraryType'}
	{attribute 'external_name' := 'F_VN_ConvertCartesianToPolarImages_GUID_EF35A358_6DCF_45B0_FB97_B9A2E5835C6F'}
	(* Converts cartesian coordinates (x, y) to polar coordinates (magnitude, angle). *)
	FUNCTION F_VN_ConvertCartesianToPolarImages : HRESULT
	VAR_INPUT
		ipSrcImageX	:	ITcVnImage;	(* Source image containing the x values (elements of type REAL or LREAL) *)
		ipSrcImageY	:	ITcVnImage;	(* Source image containing the y values (Same element type as ipSrcImageX) *)
		ipDestImageMag	:	REFERENCE TO ITcVnImage;	(* Destination image containing the magnitudes (Same element type as source images. An appropriate destination image will be created if required.) *)
		ipDestImageAng	:	REFERENCE TO ITcVnImage;	(* Destination image containing the angles (Same element type as source images. An appropriate destination image will be created if required.) *)
		hrPrev	:	HRESULT;	(* HRESULT indicating the result of previous operations (If SUCCEEDED(hrPrev) equals false, no operation is executed.) *)
	END_VAR

END_FUNCTION

// Functions/Geometric and Coordinate Transformations/F_VN_ConvertCartesianToPolarImagesExp

	{attribute 'TcIecLibraryType'}
	{attribute 'external_name' := 'F_VN_ConvertCartesianToPolarImagesExp_GUID_D044C505_06FB_441F_ECDF_74371A11C5A6'}
	(* Converts cartesian coordinates (x, y) to polar coordinates (magnitude, angle). (expert function) *)
	FUNCTION F_VN_ConvertCartesianToPolarImagesExp : HRESULT
	VAR_INPUT
		ipSrcImageX	:	ITcVnImage;	(* Source image containing the x values (elements of type REAL or LREAL) *)
		ipSrcImageY	:	ITcVnImage;	(* Source image containing the y values (Same element type as ipSrcImageX) *)
		ipDestImageMag	:	REFERENCE TO ITcVnImage;	(* Destination image containing the magnitudes (Same element type as source images. An appropriate destination image will be created if required.) *)
		ipDestImageAng	:	REFERENCE TO ITcVnImage;	(* Destination image containing the angles (Same element type as source images. An appropriate destination image will be created if required.) *)
		bAngleInDegrees	:	BOOL;	(* Specifys, if the angles should be in degrees or radians *)
		hrPrev	:	HRESULT;	(* HRESULT indicating the result of previous operations (If SUCCEEDED(hrPrev) equals false, no operation is executed.) *)
	END_VAR

END_FUNCTION

// Functions/Geometric and Coordinate Transformations/F_VN_ConvertCartesianToPolarMagnitudeImage

	{attribute 'TcIecLibraryType'}
	{attribute 'external_name' := 'F_VN_ConvertCartesianToPolarMagnitudeImage_GUID_1E0F7F07_69BF_44F5_FBC0_B5FEC64CCA11'}
	(* Converts cartesian coordinates (x, y) to polar magnitude. *)
	FUNCTION F_VN_ConvertCartesianToPolarMagnitudeImage : HRESULT
	VAR_INPUT
		ipSrcImageX	:	ITcVnImage;	(* Source image containing the x values (elements of type REAL or LREAL) *)
		ipSrcImageY	:	ITcVnImage;	(* Source image containing the y values (Same element type as ipSrcImageX) *)
		ipDestImageMag	:	REFERENCE TO ITcVnImage;	(* Destination image containing the magnitudes (Same element type as source images. An appropriate destination image will be created if required.) *)
		hrPrev	:	HRESULT;	(* HRESULT indicating the result of previous operations (If SUCCEEDED(hrPrev) equals false, no operation is executed.) *)
	END_VAR

END_FUNCTION

// Functions/Geometric and Coordinate Transformations/F_VN_ConvertCartesianToPolarMagnitudes

	{attribute 'TcIecLibraryType'}
	{attribute 'external_name' := 'F_VN_ConvertCartesianToPolarMagnitudes_GUID_00B7FCD5_9F32_4912_F52F_CFD375FE5F0F'}
	(* Converts cartesian coordinates (x, y) to polar magnitude. *)
	FUNCTION F_VN_ConvertCartesianToPolarMagnitudes : HRESULT
	VAR_INPUT
		ipSrcPointsCart	:	ITcVnContainer;	(* Container with cartesian points (ContainerType_Vector_TcVnPoint2_DINT or ContainerType_Vector_TcVnPoint2_REAL or ContainerType_Vector_TcVnPoint2_LREAL) *)
		ipDestMags	:	REFERENCE TO ITcVnContainer;	(* Returns a container which is filled with the magnitudes (ContainerType_Vector_REAL, if source points are of type TcVnPoint2_DINT or TcVnPoint2_REAL; else ContainerType_Vector_LREAL. Non-zero interface pointers are reused.) *)
		hrPrev	:	HRESULT;	(* HRESULT indicating the result of previous operations (If SUCCEEDED(hrPrev) equals false, no operation is executed.) *)
	END_VAR

END_FUNCTION

// Functions/Geometric and Coordinate Transformations/F_VN_ConvertCartesianToPolarPoints

	{attribute 'TcIecLibraryType'}
	{attribute 'external_name' := 'F_VN_ConvertCartesianToPolarPoints_GUID_0CF14846_E2D9_42D4_CD22_20B5CE2CE8AB'}
	(* Converts cartesian coordinates (x, y) to polar coordinates (magnitude, angle). *)
	FUNCTION F_VN_ConvertCartesianToPolarPoints : HRESULT
	VAR_INPUT
		ipSrcPointsCart	:	ITcVnContainer;	(* Container with cartesian points (ContainerType_Vector_TcVnPoint2_DINT or ContainerType_Vector_TcVnPoint2_REAL or ContainerType_Vector_TcVnPoint2_LREAL) *)
		ipDestPointsPolar	:	REFERENCE TO ITcVnContainer;	(* Returns a container which is filled with the converted points in polar coordinates (ContainerType_Vector_TcVnPoint2_REAL, if source points are of type TcVnPoint2_DINT or TcVnPoint2_REAL; else ContainerType_Vector_TcVnPoint2_LREAL. Non-zero interface pointers are reused.) *)
		hrPrev	:	HRESULT;	(* HRESULT indicating the result of previous operations (If SUCCEEDED(hrPrev) equals false, no operation is executed.) *)
	END_VAR

END_FUNCTION

// Functions/Geometric and Coordinate Transformations/F_VN_ConvertCartesianToPolarPointsExp

	{attribute 'TcIecLibraryType'}
	{attribute 'external_name' := 'F_VN_ConvertCartesianToPolarPointsExp_GUID_6C5EEEAD_846F_4F4C_ECF0_6F1F1D66BA8A'}
	(* Converts cartesian coordinates (x, y) to polar coordinates (magnitude, angle). (expert function) *)
	FUNCTION F_VN_ConvertCartesianToPolarPointsExp : HRESULT
	VAR_INPUT
		ipSrcPointsCart	:	ITcVnContainer;	(* Container with cartesian points (ContainerType_Vector_TcVnPoint2_DINT or ContainerType_Vector_TcVnPoint2_REAL or ContainerType_Vector_TcVnPoint2_LREAL) *)
		ipDestPointsPolar	:	REFERENCE TO ITcVnContainer;	(* Returns a container which is filled with the converted points in polar coordinates (ContainerType_Vector_TcVnPoint2_REAL, if source points are of type TcVnPoint2_DINT or TcVnPoint2_REAL; else ContainerType_Vector_TcVnPoint2_LREAL. Non-zero interface pointers are reused.) *)
		bAngleInDegrees	:	BOOL;	(* Specifys, if the angles should be in degrees or radians *)
		hrPrev	:	HRESULT;	(* HRESULT indicating the result of previous operations (If SUCCEEDED(hrPrev) equals false, no operation is executed.) *)
	END_VAR

END_FUNCTION

// Functions/Geometric and Coordinate Transformations/F_VN_ConvertPolarToCartesianImages

	{attribute 'TcIecLibraryType'}
	{attribute 'external_name' := 'F_VN_ConvertPolarToCartesianImages_GUID_C2023FF3_2784_4158_E71F_6DDE733CC7C7'}
	(* Converts polar coordinates (magnitude, angle) to cartesian coordinates (x, y). *)
	FUNCTION F_VN_ConvertPolarToCartesianImages : HRESULT
	VAR_INPUT
		ipSrcImageMag	:	ITcVnImage;	(* Source image containing the magnitudes (elements of type REAL or LREAL) *)
		ipSrcImageAng	:	ITcVnImage;	(* Source image containing the angles (Same element type as ipSrcImageMag) *)
		ipDestImageX	:	REFERENCE TO ITcVnImage;	(* Destination image containing the x values (Same element type as source images. An appropriate destination image will be created if required.) *)
		ipDestImageY	:	REFERENCE TO ITcVnImage;	(* Destination image containing the y values (Same element type as source images. An appropriate destination image will be created if required.) *)
		hrPrev	:	HRESULT;	(* HRESULT indicating the result of previous operations (If SUCCEEDED(hrPrev) equals false, no operation is executed.) *)
	END_VAR

END_FUNCTION

// Functions/Geometric and Coordinate Transformations/F_VN_ConvertPolarToCartesianImagesExp

	{attribute 'TcIecLibraryType'}
	{attribute 'external_name' := 'F_VN_ConvertPolarToCartesianImagesExp_GUID_9D55688F_950A_4A67_D579_DE992620A88A'}
	(* Converts polar coordinates (magnitude, angle) to cartesian coordinates (x, y). (expert function) *)
	FUNCTION F_VN_ConvertPolarToCartesianImagesExp : HRESULT
	VAR_INPUT
		ipSrcImageMag	:	ITcVnImage;	(* Source image containing the magnitudes (elements of type REAL or LREAL) *)
		ipSrcImageAng	:	ITcVnImage;	(* Source image containing the angles (Same element type as ipSrcImageMag) *)
		ipDestImageX	:	REFERENCE TO ITcVnImage;	(* Destination image containing the x values (Same element type as source images. An appropriate destination image will be created if required.) *)
		ipDestImageY	:	REFERENCE TO ITcVnImage;	(* Destination image containing the y values (Same element type as source images. An appropriate destination image will be created if required.) *)
		bAngleInDegrees	:	BOOL;	(* Specifys, if the angles are in degrees or radians *)
		hrPrev	:	HRESULT;	(* HRESULT indicating the result of previous operations (If SUCCEEDED(hrPrev) equals false, no operation is executed.) *)
	END_VAR

END_FUNCTION

// Functions/Geometric and Coordinate Transformations/F_VN_ConvertPolarToCartesianPoints

	{attribute 'TcIecLibraryType'}
	{attribute 'external_name' := 'F_VN_ConvertPolarToCartesianPoints_GUID_4A79B0D6_1CFC_4B15_D047_28F1CAC5F597'}
	(* Converts polar coordinates (magnitude, angle) to cartesian coordinates (x, y). *)
	FUNCTION F_VN_ConvertPolarToCartesianPoints : HRESULT
	VAR_INPUT
		ipSrcPointsPolar	:	ITcVnContainer;	(* Container with polar coordinates (ContainerType_Vector_TcVnPoint2_REAL or ContainerType_Vector_TcVnPoint2_LREAL) *)
		ipDestPointsCart	:	REFERENCE TO ITcVnContainer;	(* Returns a container which is filled with the converted points in cartesian coordinates (same type ID as ipSrcPointsPolar. Non-zero interface pointers are reused.) *)
		hrPrev	:	HRESULT;	(* HRESULT indicating the result of previous operations (If SUCCEEDED(hrPrev) equals false, no operation is executed.) *)
	END_VAR

END_FUNCTION

// Functions/Geometric and Coordinate Transformations/F_VN_ConvertPolarToCartesianPointsExp

	{attribute 'TcIecLibraryType'}
	{attribute 'external_name' := 'F_VN_ConvertPolarToCartesianPointsExp_GUID_166FEFE1_269F_4A28_DAB0_A444B33EFE5E'}
	(* Converts polar coordinates (magnitude, angle) to cartesian coordinates (x, y). (expert function) *)
	FUNCTION F_VN_ConvertPolarToCartesianPointsExp : HRESULT
	VAR_INPUT
		ipSrcPointsPolar	:	ITcVnContainer;	(* Container with polar coordinates (ContainerType_Vector_TcVnPoint2_REAL or ContainerType_Vector_TcVnPoint2_LREAL) *)
		ipDestPointsCart	:	REFERENCE TO ITcVnContainer;	(* Returns a container which is filled with the converted points in cartesian coordinates (same type ID as ipSrcPointsPolar. Non-zero interface pointers are reused.) *)
		bAngleInDegrees	:	BOOL;	(* Specifys, if the angles are in degrees or radians *)
		hrPrev	:	HRESULT;	(* HRESULT indicating the result of previous operations (If SUCCEEDED(hrPrev) equals false, no operation is executed.) *)
	END_VAR

END_FUNCTION

// Functions/Geometric and Coordinate Transformations/F_VN_DecomposeAffineTransformation

	{attribute 'TcIecLibraryType'}
	{attribute 'external_name' := 'F_VN_DecomposeAffineTransformation_GUID_1F356C85_2073_44A1_D001_E5E9DA7C502C'}
	(* Decompose an affine transformation matrix and return the rotation angle (clockwise) in radian. The decomposition method assumes the following order of transformation: Translation, Rotation, Scale, and Skew. *)
	FUNCTION F_VN_DecomposeAffineTransformation : HRESULT
	VAR_IN_OUT
		aAffineTransform	:	TcVnMatrix2x3_LREAL;	(* Affine transformation matrix *)
		fRotationAngle	:	LREAL;	(* Rotation angle (radian) in the clockwise direction. The rotation center is the origin point (0,0) *)
	END_VAR
	VAR_INPUT
		hrPrev	:	HRESULT;	(* HRESULT indicating the result of previous operations (If SUCCEEDED(hrPrev) equals false, no operation is executed.) *)
	END_VAR

END_FUNCTION

// Functions/Geometric and Coordinate Transformations/F_VN_DecomposeAffineTransformationExp

	{attribute 'TcIecLibraryType'}
	{attribute 'external_name' := 'F_VN_DecomposeAffineTransformationExp_GUID_1D961019_3976_4822_FD82_36BCEE30E5BD'}
	(* Decompose an affine transformation matrix and return the rotation angle (clockwise) in radian, translation vector (pixels), scale, and skew vectors (angle in radian). The decomposition method assumes the following order of transformation: Translation, Rotation, Scale, and Skew. *)
	FUNCTION F_VN_DecomposeAffineTransformationExp : HRESULT
	VAR_IN_OUT
		aAffineTransform	:	TcVnMatrix2x3_LREAL;	(* Affine transformation matrix *)
		fRotationAngle	:	LREAL;	(* Rotation angle (radian) in the clockwise direction. The rotation center is the origin point (0,0) *)
		aTranslationVector	:	TcVnVector2_LREAL;	(* 2D translation vector. The values are in pixels *)
		aScaleVector	:	TcVnVector2_LREAL;	(* 2D scale vector  *)
		aSkewVector	:	TcVnVector2_LREAL;	(* 2D skew vector. The values are the skew angles in x and y directions in radian *)
	END_VAR
	VAR_INPUT
		hrPrev	:	HRESULT;	(* HRESULT indicating the result of previous operations (If SUCCEEDED(hrPrev) equals false, no operation is executed.) *)
	END_VAR

END_FUNCTION

// Functions/Geometric and Coordinate Transformations/F_VN_DecomposeHomography

	{attribute 'TcIecLibraryType'}
	{attribute 'external_name' := 'F_VN_DecomposeHomography_GUID_1F10B58D_BB13_48D9_FE45_9365CA0D370F'}
	(* Decompose a homography matrix into four solutions of rotation, translation, and plane normal. It returns two solutions (Ra, Ta, Nb) and (Rb, Tb, Nb). The third and the fourth solutions can be calculated as follows: (Ra, -Ta, -Na) and (Rb, -Tb, -Nb). *)
	FUNCTION F_VN_DecomposeHomography : HRESULT
	VAR_IN_OUT
		aHomography	:	TcVnMatrix3x3_LREAL;	(* Homography matrix (a perspective transformation between two planes) *)
		aCameraMatrix	:	TcVnMatrix3x3_LREAL;	(* Camera matrix *)
		aRotationMatrixA	:	TcVnMatrix3x3_LREAL;	(* Rotation matrix of the first solution (Ra) *)
		aTranslationVectorA	:	TcVnVector3_LREAL;	(* Translation vector of the first solution (Ta) *)
		aNormVectorA	:	TcVnVector3_LREAL;	(* Norm vector of the first solution (Na) *)
		aRotationMatrixB	:	TcVnMatrix3x3_LREAL;	(* Rotation matrix of the second solution (Rb) *)
		aTranslationVectorB	:	TcVnVector3_LREAL;	(* Translation vector of the second solution (Tb) *)
		aNormVectorB	:	TcVnVector3_LREAL;	(* Norm vector of the second solution Nb *)
	END_VAR
	VAR_INPUT
		hrPrev	:	HRESULT;	(* HRESULT indicating the result of previous operations (If SUCCEEDED(hrPrev) equals false, no operation is executed.) *)
	END_VAR
	VAR_OUTPUT
		nSolutions	:	UDINT;	(* Returns the number of solutions. In normal cases, it is equal four.  *)
	END_VAR

END_FUNCTION

// Functions/Geometric and Coordinate Transformations/F_VN_DecomposeHomographyExp

	{attribute 'TcIecLibraryType'}
	{attribute 'external_name' := 'F_VN_DecomposeHomographyExp_GUID_63B3E845_574B_44DD_FF11_70BF8A6FAEA1'}
	(* Decompose a homography matrix and verify four solutions of rotation, translation, and plane normal. It uses visible reference points being in front of the camera to confirm which solution(s) of the four solutions (maximum two solutions) are consistent with all reference points. *)
	FUNCTION F_VN_DecomposeHomographyExp : HRESULT
	VAR_IN_OUT
		aHomography	:	TcVnMatrix3x3_LREAL;	(* Homography matrix (a perspective transformation between two planes) *)
		aCameraMatrix	:	TcVnMatrix3x3_LREAL;	(* Camera matrix *)
		aRotationMatrixA	:	TcVnMatrix3x3_LREAL;	(* Rotation matrix of the first solution (Ra) *)
		aTranslationVectorA	:	TcVnVector3_LREAL;	(* Translation vector of the first solution (Ta) *)
		aNormVectorA	:	TcVnVector3_LREAL;	(* Norm vector of the first solution (Na) *)
		aRotationMatrixB	:	TcVnMatrix3x3_LREAL;	(* Rotation matrix of the second solution (Rb) *)
		aTranslationVectorB	:	TcVnVector3_LREAL;	(* Translation vector of the second solution (Tb) *)
		aNormVectorB	:	TcVnVector3_LREAL;	(* Norm vector of the second solution (Nb) *)
	END_VAR
	VAR_INPUT
		ipPointsSrc	:	ITcVnContainer;	(* Container with source points (ContainerType_Vector_TcVnPoint2_REAL) *)
		ipPointsDes	:	ITcVnContainer;	(* Container with destination points (same number as ipPoints1, ContainerType_Vector_TcVnPoint2_REAL) *)
		ipInlierMask	:	ITcVnContainer;	(* A mask marking the inliers (optional, set to 0 if not available; ContainerType_Vector_SINT or ContainerType_Vector_USINT) *)
		hrPrev	:	HRESULT;	(* HRESULT indicating the result of previous operations (If SUCCEEDED(hrPrev) equals false, no operation is executed.) *)
	END_VAR
	VAR_OUTPUT
		nSolutions	:	UDINT;	(* Return the number of true potential solutions [0,1, or 2].
							0: no true potential solutions for the given corresponding points are confirmed.
							1: the solution (Ra, Ta, Na) is confirmed.
							2: both solution (Ra, Ta, Na) and (Rb, Tb, Nb) are confirmed.
							In all cases the function returns two solutions (Ra, Ta, Nb) and (Rb, Tb, Nb). The third and the fourth solutions can be calculated as follows: (Ra, -Ta, -Na) and (Rb, -Tb, -Nb).
						 *)
	END_VAR

END_FUNCTION

// Functions/Geometric and Coordinate Transformations/F_VN_FlipImage

	{attribute 'TcIecLibraryType'}
	{attribute 'external_name' := 'F_VN_FlipImage_GUID_CF5381B5_C061_4CE7_FE8E_B48DD5F55808'}
	(* Flip an image (mirror and shift back to prior coordinates). *)
	FUNCTION F_VN_FlipImage : HRESULT
	VAR_INPUT
		ipSrcImage	:	ITcVnImage;	(* Source image *)
		ipDestImage	:	REFERENCE TO ITcVnImage;	(* Destination image (An appropriate destination image will be created if required.) *)
		eFlipAxis	:	ETcVnFlipAxis;	(* Selects the axis around which to flip the image *)
		hrPrev	:	HRESULT;	(* HRESULT indicating the result of previous operations (If SUCCEEDED(hrPrev) equals false, no operation is executed.) *)
	END_VAR

END_FUNCTION

// Functions/Geometric and Coordinate Transformations/F_VN_GenerateAffineTransformationUnitMatrix2D

	{attribute 'TcIecLibraryType'}
	{attribute 'external_name' := 'F_VN_GenerateAffineTransformationUnitMatrix2D_GUID_8996CF80_E37D_42D6_F9F8_2516071FF612'}
	(* Generate an affine transformation 2D unit matrix. *)
	FUNCTION F_VN_GenerateAffineTransformationUnitMatrix2D : HRESULT
	VAR_IN_OUT
		aTransformationMatrix	:	TcVnMatrix2x3_LREAL;	(* Resulting affine transformation unit matrix *)
	END_VAR
	VAR_INPUT
		hrPrev	:	HRESULT;	(* HRESULT indicating the result of previous operations (If SUCCEEDED(hrPrev) equals false, no operation is executed.) *)
	END_VAR

END_FUNCTION

// Functions/Geometric and Coordinate Transformations/F_VN_GetAffineTransformation

	{attribute 'TcIecLibraryType'}
	{attribute 'external_name' := 'F_VN_GetAffineTransformation_GUID_F874DA6B_6668_4679_FD89_8F08A440EABE'}
	(* Calculate the affine transformation between three corresponding point pairs. The points mark the corners of the corresponding triangles. *)
	FUNCTION F_VN_GetAffineTransformation : HRESULT
	VAR_IN_OUT
		aSrcPoints	:	TcVnArray3_Point2_REAL;	(* Source points *)
		aDestPoints	:	TcVnArray3_Point2_REAL;	(* Destination points *)
		aTransformationMatrix	:	TcVnMatrix2x3_LREAL;	(* Resulting transformation matrix *)
	END_VAR
	VAR_INPUT
		hrPrev	:	HRESULT;	(* HRESULT indicating the result of previous operations (If SUCCEEDED(hrPrev) equals false, no operation is executed.) *)
	END_VAR

END_FUNCTION

// Functions/Geometric and Coordinate Transformations/F_VN_GetAffineTransformation2D

	{attribute 'TcIecLibraryType'}
	{attribute 'external_name' := 'F_VN_GetAffineTransformation2D_GUID_F22F1852_E9BB_4FED_F3D4_2AAA139564A2'}
	(* Estimate the 2D affine transformation between two planar point sets using RANSAC algorithm. *)
	FUNCTION F_VN_GetAffineTransformation2D : HRESULT
	VAR_INPUT
		ipSrcPoints	:	ITcVnContainer;	(* Container with at least 3 source points (ContainerType_Vector_TcVnPoint2_REAL) *)
		ipDestPoints	:	ITcVnContainer;	(* Container with destination points (same number as ipSrcPoints, ContainerType_Vector_TcVnPoint2_REAL) *)
	END_VAR
	VAR_IN_OUT
		aAffineTransform	:	TcVnMatrix2x3_LREAL;	(* Returns the affine transformation matrix, which transforms the source points to the destination points *)
	END_VAR
	VAR_INPUT
		hrPrev	:	HRESULT;	(* HRESULT indicating the result of previous operations (If SUCCEEDED(hrPrev) equals false, no operation is executed.) *)
	END_VAR

END_FUNCTION

// Functions/Geometric and Coordinate Transformations/F_VN_GetAffineTransformation2DExp

	{attribute 'TcIecLibraryType'}
	{attribute 'external_name' := 'F_VN_GetAffineTransformation2DExp_GUID_20CE1F02_E27E_4CF2_FDC7_DF9853CDBB21'}
	(* Estimate the affine transformation between two planar point sets. (expert function) *)
	FUNCTION F_VN_GetAffineTransformation2DExp : HRESULT
	VAR_INPUT
		ipSrcPoints	:	ITcVnContainer;	(* Container with at least 3 source points (ContainerType_Vector_TcVnPoint2_REAL) *)
		ipDestPoints	:	ITcVnContainer;	(* Container with destination points (same number as ipSrcPoints, ContainerType_Vector_TcVnPoint2_REAL) *)
	END_VAR
	VAR_IN_OUT
		aAffineTransform	:	TcVnMatrix2x3_LREAL;	(* Returns the affine transformation matrix, which transforms the source points to the destination points *)
	END_VAR
	VAR_INPUT
		eAlgorithm	:	ETcVnEstimationAlgorithm;	(* Estimation algorithm (only RANSAC and LMEDS are supported) *)
		fReprojThreshold	:	LREAL;	(* Maximum allowed reprojection error to treat a point pair as an inlier *)
		ipInlierMask	:	REFERENCE TO ITcVnContainer;	(* Returns a mask marking the inliers (optional, set to 0 if not required; ContainerType_Vector_USINT) *)
		nMaxIterations	:	UDINT;	(* Maximum number of iterations *)
		fConfidence	:	LREAL;	(* Confidence (0..1) *)
		nRefineIters	:	UDINT;	(* Maximum number of iterations of Levenberg-Marquardt algorithm to refine further the affine transform (using only inliers). Set to 0 to disable refining. *)
		hrPrev	:	HRESULT;	(* HRESULT indicating the result of previous operations (If SUCCEEDED(hrPrev) equals false, no operation is executed.) *)
	END_VAR

END_FUNCTION

// Functions/Geometric and Coordinate Transformations/F_VN_GetPerspectiveTransformation

	{attribute 'TcIecLibraryType'}
	{attribute 'external_name' := 'F_VN_GetPerspectiveTransformation_GUID_749A872C_16DC_466E_DA6D_5B2CA09D7D73'}
	(* Calculate the perspective transformation between four corresponding point pairs. The points mark the corners of the corresponding rectangles. *)
	FUNCTION F_VN_GetPerspectiveTransformation : HRESULT
	VAR_IN_OUT
		aSrcPoints	:	TcVnArray4_Point2_REAL;	(* Source points *)
		aDestPoints	:	TcVnArray4_Point2_REAL;	(* Destination points *)
		aTransformationMatrix	:	TcVnMatrix3x3_LREAL;	(* Resulting transformation matrix *)
	END_VAR
	VAR_INPUT
		hrPrev	:	HRESULT;	(* HRESULT indicating the result of previous operations (If SUCCEEDED(hrPrev) equals false, no operation is executed.) *)
	END_VAR

END_FUNCTION

// Functions/Geometric and Coordinate Transformations/F_VN_Homography

	{attribute 'TcIecLibraryType'}
	{attribute 'external_name' := 'F_VN_Homography_GUID_0A5AE478_2FBD_480E_EA03_ED46DF1154BC'}
	(* Find the homography (perspective transformation) between two planar point sets using RANSAC algorithm. *)
	FUNCTION F_VN_Homography : HRESULT
	VAR_INPUT
		ipSrcPoints	:	ITcVnContainer;	(* Container with at least 4 source points (ContainerType_Vector_TcVnPoint2_REAL) *)
		ipDestPoints	:	ITcVnContainer;	(* Container with destination points (same number as ipSrcPoints, ContainerType_Vector_TcVnPoint2_REAL) *)
	END_VAR
	VAR_IN_OUT
		aPerspectiveTransform	:	TcVnMatrix3x3_LREAL;	(* Returns the perspective transformation matrix, which transforms the source points to the destination points *)
	END_VAR
	VAR_INPUT
		hrPrev	:	HRESULT;	(* HRESULT indicating the result of previous operations (If SUCCEEDED(hrPrev) equals false, no operation is executed.) *)
	END_VAR

END_FUNCTION

// Functions/Geometric and Coordinate Transformations/F_VN_HomographyExp

	{attribute 'TcIecLibraryType'}
	{attribute 'external_name' := 'F_VN_HomographyExp_GUID_25EFF2D2_F8C5_49CC_D571_A962D9615AEB'}
	(* Find the homography (perspective transformation) between two planar point sets. (expert function) *)
	FUNCTION F_VN_HomographyExp : HRESULT
	VAR_INPUT
		ipSrcPoints	:	ITcVnContainer;	(* Container with at least 4 source points (ContainerType_Vector_TcVnPoint2_REAL) *)
		ipDestPoints	:	ITcVnContainer;	(* Container with destination points (same number as ipSrcPoints, ContainerType_Vector_TcVnPoint2_REAL) *)
	END_VAR
	VAR_IN_OUT
		aPerspectiveTransform	:	TcVnMatrix3x3_LREAL;	(* Returns the perspective transformation matrix, which transforms the source points to the destination points *)
	END_VAR
	VAR_INPUT
		eAlgorithm	:	ETcVnEstimationAlgorithm;	(* Estimation algorithm *)
		fReprojThreshold	:	LREAL;	(* Maximum allowed reprojection error to treat a point pair as an inlier (only for RANSAC, RHO) *)
		ipInlierMask	:	REFERENCE TO ITcVnContainer;	(* Returns a mask marking the inliers (optional, set to 0 if not required; ContainerType_Vector_SINT; only for RANSAC, LMEDS) *)
		nMaxIterations	:	UDINT;	(* Maximum number of RANSAC iterations *)
		fConfidence	:	LREAL;	(* Confidence (0..1) *)
		hrPrev	:	HRESULT;	(* HRESULT indicating the result of previous operations (If SUCCEEDED(hrPrev) equals false, no operation is executed.) *)
	END_VAR

END_FUNCTION

// Functions/Geometric and Coordinate Transformations/F_VN_InvertAffineTransformation

	{attribute 'TcIecLibraryType'}
	{attribute 'external_name' := 'F_VN_InvertAffineTransformation_GUID_2C470677_2E35_4074_DA25_EEE617817764'}
	(* Invert a 2D affine transformation matrix. The inverted transformation compensates the affine transformation on an image if it is used in the F_VN_WarpAffine function. *)
	FUNCTION F_VN_InvertAffineTransformation : HRESULT
	VAR_IN_OUT
		aTransformationMatrix	:	TcVnMatrix2x3_LREAL;	(* Source affine transformation matrix *)
		aInvertedTransformationMatrix	:	TcVnMatrix2x3_LREAL;	(* Resulting inverted affine transformation matrix *)
	END_VAR
	VAR_INPUT
		hrPrev	:	HRESULT;	(* HRESULT indicating the result of previous operations (If SUCCEEDED(hrPrev) equals false, no operation is executed.) *)
	END_VAR

END_FUNCTION

// Functions/Geometric and Coordinate Transformations/F_VN_WarpAffine

	{attribute 'TcIecLibraryType'}
	{attribute 'external_name' := 'F_VN_WarpAffine_GUID_9792240A_C94E_4415_FA9E_0FB7C68DF254'}
	(* Apply an affine transformation to an image. *)
	FUNCTION F_VN_WarpAffine : HRESULT
	VAR_INPUT
		ipSrcImage	:	ITcVnImage;	(* Source image *)
		ipDestImage	:	REFERENCE TO ITcVnImage;	(* Destination image (An appropriate image will be created if required.) *)
	END_VAR
	VAR_IN_OUT
		aTransformationMatrix	:	TcVnMatrix2x3_LREAL;	(* Affine transformation matrix *)
	END_VAR
	VAR_INPUT
		hrPrev	:	HRESULT;	(* HRESULT indicating the result of previous operations (If SUCCEEDED(hrPrev) equals false, no operation is executed.) *)
	END_VAR

END_FUNCTION

// Functions/Geometric and Coordinate Transformations/F_VN_PerspectiveTransformation

	{attribute 'TcIecLibraryType'}
	{attribute 'external_name' := 'F_VN_PerspectiveTransformation_GUID_119F1E65_BAAA_4841_D6BB_057BB17D5958'}
	(* Apply a perspective transformation (rotation + translation, e.g. from extrinsic calibration) to 3D point coordinates. *)
	FUNCTION F_VN_PerspectiveTransformation : HRESULT
	VAR_INPUT
		ipSrcPoints	:	ITcVnContainer;	(* Container with 3D source points (TcVnPoint3_REAL or TcVnPoint3_LREAL) *)
		ipDestPoints	:	REFERENCE TO ITcVnContainer;	(* Returns the transformed points (same type as ipSrcPoints) *)
	END_VAR
	VAR_IN_OUT
		aRotationMatrix	:	TcVnMatrix3x3_LREAL;	(* 3x3 rotation matrix *)
		aTranslationVector	:	TcVnVector3_LREAL;	(* Translation vector *)
	END_VAR
	VAR_INPUT
		hrPrev	:	HRESULT;	(* HRESULT indicating the result of previous operations (If SUCCEEDED(hrPrev) equals false, no operation is executed.) *)
	END_VAR

END_FUNCTION

// Functions/Geometric and Coordinate Transformations/F_VN_PyramidDown

	{attribute 'TcIecLibraryType'}
	{attribute 'external_name' := 'F_VN_PyramidDown_GUID_14F8FC87_76F4_4A8E_CBDF_2421E498D097'}
	(* Downsamples an image to half width and height. *)
	FUNCTION F_VN_PyramidDown : HRESULT
	VAR_INPUT
		ipSrcImage	:	ITcVnImage;	(* Source image *)
		ipDestImage	:	REFERENCE TO ITcVnImage;	(* Destination image (An appropriate destination image will be created if required.) *)
		hrPrev	:	HRESULT;	(* HRESULT indicating the result of previous operations (If SUCCEEDED(hrPrev) equals false, no operation is executed.) *)
	END_VAR

END_FUNCTION

// Functions/Geometric and Coordinate Transformations/F_VN_PyramidUp

	{attribute 'TcIecLibraryType'}
	{attribute 'external_name' := 'F_VN_PyramidUp_GUID_77F6F96E_EE98_4CEA_D306_94A555B173ED'}
	(* Upsamples an image to double width and height. *)
	FUNCTION F_VN_PyramidUp : HRESULT
	VAR_INPUT
		ipSrcImage	:	ITcVnImage;	(* Source image *)
		ipDestImage	:	REFERENCE TO ITcVnImage;	(* Destination image (An appropriate destination image will be created if required.) *)
		hrPrev	:	HRESULT;	(* HRESULT indicating the result of previous operations (If SUCCEEDED(hrPrev) equals false, no operation is executed.) *)
	END_VAR

END_FUNCTION

// Functions/Geometric and Coordinate Transformations/F_VN_RemapImageToLogPolarSpace

	{attribute 'TcIecLibraryType'}
	{attribute 'external_name' := 'F_VN_RemapImageToLogPolarSpace_GUID_81EA7AEF_CBC9_4D3E_E6C3_0229A0E4604E'}
	(* Remap an image to log-polar space. *)
	FUNCTION F_VN_RemapImageToLogPolarSpace : HRESULT
	VAR_INPUT
		ipSrcImage	:	ITcVnImage;	(* Source image *)
		ipDestImage	:	REFERENCE TO ITcVnImage;	(* Destination image (Must not be the same as ipSrcImage! An appropriate destination image will be created if required.) *)
	END_VAR
	VAR_IN_OUT
		aCenter	:	TcVnPoint2_REAL;	(* Center point for the transformation *)
	END_VAR
	VAR_INPUT
		hrPrev	:	HRESULT;	(* HRESULT indicating the result of previous operations (If SUCCEEDED(hrPrev) equals false, no operation is executed.) *)
	END_VAR

END_FUNCTION

// Functions/Geometric and Coordinate Transformations/F_VN_RemapImageToLogPolarSpaceExp

	{attribute 'TcIecLibraryType'}
	{attribute 'external_name' := 'F_VN_RemapImageToLogPolarSpaceExp_GUID_74C60EB8_8785_4F75_D016_41EE6A7F61DB'}
	(* Remap an image to log-polar space. (expert function) *)
	FUNCTION F_VN_RemapImageToLogPolarSpaceExp : HRESULT
	VAR_INPUT
		ipSrcImage	:	ITcVnImage;	(* Source image *)
		ipDestImage	:	REFERENCE TO ITcVnImage;	(* Destination image (Must not be the same as ipSrcImage! An appropriate destination image will be created if required.) *)
	END_VAR
	VAR_IN_OUT
		aCenter	:	TcVnPoint2_REAL;	(* Center point for the transformation *)
	END_VAR
	VAR_INPUT
		fScale	:	LREAL;	(* Magnitude scale parameter, i.e. image width / ln(radius) (set to 0 for auto select) *)
		eInterpolationType	:	ETcVnInterpolationType;	(* Interpolation type *)
		hrPrev	:	HRESULT;	(* HRESULT indicating the result of previous operations (If SUCCEEDED(hrPrev) equals false, no operation is executed.) *)
	END_VAR

END_FUNCTION

// Functions/Geometric and Coordinate Transformations/F_VN_RemapImageToLogPolarSpaceExp2

	{attribute 'TcIecLibraryType'}
	{attribute 'external_name' := 'F_VN_RemapImageToLogPolarSpaceExp2_GUID_3C34428E_2799_4AD4_F2CA_DE30BE238784'}
	(* Remap an image to log-polar space. (expert function) *)
	FUNCTION F_VN_RemapImageToLogPolarSpaceExp2 : HRESULT
	VAR_INPUT
		ipSrcImage	:	ITcVnImage;	(* Source image *)
		ipDestImage	:	REFERENCE TO ITcVnImage;	(* Destination image (Must not be the same as ipSrcImage! An appropriate destination image will be created if required.) *)
	END_VAR
	VAR_IN_OUT
		aCenter	:	TcVnPoint2_REAL;	(* Center point for the transformation *)
	END_VAR
	VAR_INPUT
		fScale	:	LREAL;	(* Magnitude scale parameter, i.e. image width / ln(radius) (set to 0 for auto select) *)
		eInterpolationType	:	ETcVnInterpolationType;	(* Interpolation type *)
		nDestWidth	:	DINT;	(* Destination image width (set to -1 for source image width, 0 to auto scale to transformed radius, > 0 for a user defined width) *)
		nDestHeight	:	DINT;	(* destination image height (set to -1 for source image height, 0 to auto scale to transformed radius * PI, > 0 for a user defined height) *)
		hrPrev	:	HRESULT;	(* HRESULT indicating the result of previous operations (If SUCCEEDED(hrPrev) equals false, no operation is executed.) *)
	END_VAR

END_FUNCTION

// Functions/Geometric and Coordinate Transformations/F_VN_RemapImageToPolarSpace

	{attribute 'TcIecLibraryType'}
	{attribute 'external_name' := 'F_VN_RemapImageToPolarSpace_GUID_31360372_C224_4667_E7DE_1CB0BFAFBB50'}
	(* Remap an image to polar space. *)
	FUNCTION F_VN_RemapImageToPolarSpace : HRESULT
	VAR_INPUT
		ipSrcImage	:	ITcVnImage;	(* Source image *)
		ipDestImage	:	REFERENCE TO ITcVnImage;	(* Destination image (Must not be the same as ipSrcImage! An appropriate destination image will be created if required.) *)
	END_VAR
	VAR_IN_OUT
		aCenter	:	TcVnPoint2_REAL;	(* Center point for the transformation *)
	END_VAR
	VAR_INPUT
		hrPrev	:	HRESULT;	(* HRESULT indicating the result of previous operations (If SUCCEEDED(hrPrev) equals false, no operation is executed.) *)
	END_VAR

END_FUNCTION

// Functions/Geometric and Coordinate Transformations/F_VN_RemapImageToPolarSpaceExp

